				BESTUECKZELLE_1720:
					fb_state_entry.i16_next_step := 40;
			END_CASE
		END_IF

(*=======================================================*)
	35:	(* CAM OUT Y-Achse *)
		IF fb_state_entry.E THEN
			st_drive_cmd_y_achse.enu_cmd := CAM_OUT_SLAVE;
		END_IF

		(*-----------------------Weiterschaltbedingungen----------------------------*)
		IF st_drive_cmd_y_achse.enu_cmd = NO_COMMAND AND NOT fb_state_entry.E THEN
			fb_state_entry.i16_next_step := 40;
		END_IF

(*=======================================================*)
	40:	(* Reglerfreigabe setzen , Reset wird bei Bedarf automatisch ausgeführt*)
		IF fb_state_entry.E THEN
			st_drive_cmd.enu_cmd := POWER_ENABLE;
		END_IF

		(*-----------------------Weiterschaltbedingungen----------------------------*)
		IF st_drive_cmd.enu_cmd = NO_COMMAND THEN
			fb_state_entry.i16_next_step := 50;
		END_IF

(*=======================================================*)
	50:	(* Nullpunktverschiebung ist geschrieben *)
		IF fb_state_entry.E THEN
			st_ctrl_out.b_prebereit := TRUE;
		END_IF

		(*-----------------------Weiterschaltbedingungen----------------------------*)
		IF st_ctrl_in.b_init THEN
			CASE gst_datensatz.st_md.i16_typ_zelle OF
				KEINE_ZELLE:
					;

				BESTUECKZELLE_1700, RASTERFOLIE:
					fb_state_entry.i16_next_step := 60;

				BESTUECKZELLE_1720:
					fb_state_entry.i16_next_step := 95;
			END_CASE
		END_IF

(*=======================================================*)
	60: (* Abfrage der Positionen von Z-Achse und Y-Achse *)

		(*-----------------------Weiterschaltbedingungen----------------------------*)
		IF 	z_achse.NcToPlc.ActPos > ST_MotionFunctionPoints.YZTischMasterPos3 AND
			ABS(y_achse.NcToPlc.ActPos - gst_datensatz.st_md.st_md_y_achse.lr_wt_uebergabepos) > 0.5
			THEN
				(* Y-Achse steht in Kollision mit Antriebskonus des Förderbands *)
				fb_state_entry.i16_next_step := 70;
		ELSE
			i16_kollisionszaehler := 0;
			fb_state_entry.i16_next_step := 80;
		END_IF

(*=======================================================*)
	70: (* Im Wiederhohlungsfall -> Fehler *)
		IF fb_state_entry.E THEN
			i16_kollisionszaehler := i16_kollisionszaehler + 1;
		END_IF

		(*-----------------------Weiterschaltbedingungen----------------------------*)
		IF i16_kollisionszaehler > 1 THEN
			sm_positionsueberwachung := TRUE;
			fb_state_entry.i16_next_step := FEHLER;
		ELSE
			fb_state_entry.i16_next_step := 75;
		END_IF

(*=======================================================*)
	75:	(* Fahre Z-Achse und damit Y-Achse aus der Kollisionsposition *)
		IF fb_state_entry.E THEN
			fb_axis.lr_soll_geschwindigkeit := gst_datensatz.st_wkz.r_auto_z;
			fb_axis.st_position.r_soll := ST_MotionFunctionPoints.YZTischMasterPos3;
			st_drive_cmd.enu_cmd := MOVE_ABSOLUTE;
		END_IF

		(*-----------------------Weiterschaltbedingungen----------------------------*)
		IF st_drive_cmd.enu_cmd = NO_COMMAND THEN
			fb_state_entry.i16_next_step := 80;
		END_IF

(*=======================================================*)
	80: (* Auslesen der Y-Position an der aktuellen Z-Position in der Kurvenscheibe *)
		IF fb_state_entry.E THEN
			fb_axis_y_achse.r_master_position := z_achse.NcToPlc.ActPos;
			st_drive_cmd_y_achse.enu_cmd := READ_SLAVE_DYNAMICS;
		END_IF

		(*-----------------------Weiterschaltbedingungen----------------------------*)
		IF st_drive_cmd_y_achse.enu_cmd = NO_COMMAND AND NOT fb_state_entry.E THEN
			fb_state_entry.i16_next_step := 85;
		END_IF

(*=======================================================*)
	85: (* Starte Y-Achse auf die entsprechende Position in der Kurvenscheibe *)
		IF fb_state_entry.E THEN
			lr_slave_position := fb_axis_y_achse.mc_read_camtable_slave_dynamics.SlavePosition;
			axis_y_achse.st_ctrl.in.b_start := TRUE;
		END_IF

		(*-----------------------Weiterschaltbedingungen----------------------------*)
		IF axis_y_achse.st_ctrl.out.b_fertig AND NOT fb_state_entry.E THEN
			axis_y_achse.st_ctrl.in.b_start := FALSE;
			fb_state_entry.i16_next_step := 90;
		END_IF

(*=======================================================*)
	90:	(* CAM IN Y-Achse *)
		IF fb_state_entry.E THEN
			fb_axis_y_achse.st_camscaling_data.SlaveScaling := 1;
			st_drive_cmd_y_achse.enu_cmd := CAM_IN_SLAVE;
		END_IF

		IF y_achse.NcToPlc.CoupleState = 0 THEN
			st_drive_cmd_y_achse.enu_cmd := CAM_IN_SLAVE;
		END_IF

		(*-----------------------Weiterschaltbedingungen----------------------------*)
		IF st_drive_cmd_y_achse.enu_cmd = NO_COMMAND AND NOT fb_state_entry.E THEN
			fb_state_entry.i16_next_step := 95;
		END_IF

(*=======================================================*)
	95:	(* Fahre Z-Achse auf die WT-Übergabeposition *)
		IF fb_state_entry.E THEN
			fb_axis.lr_soll_geschwindigkeit := gst_datensatz.st_wkz.r_auto_z;
			fb_axis.st_position.r_soll := gst_datensatz.st_md.st_md_z_achse.lr_wt_uebergabepos;
			st_drive_cmd.enu_cmd := MOVE_ABSOLUTE;
		END_IF

		(*-----------------------Weiterschaltbedingungen----------------------------*)
		IF st_drive_cmd.enu_cmd = NO_COMMAND THEN
			fb_state_entry.i16_next_step := BEREIT;
		END_IF

(*=======================================================*)
	BEREIT:
		IF fb_state_entry.E THEN
			st_ctrl_out.b_busy:=FALSE;
			st_ctrl_out.b_bereit := TRUE;
			st_ctrl_out.b_fertig := TRUE;
			bm_rastnasen_1_fehlt := FALSE;
			bm_rastnasen_2_fehlt := FALSE;
			enu_cmd_in:=NO_COMMAND;
		END_IF

		IF NOT gst_datensatz.st_wkz.b_rafo_auto_einf_aktiv THEN
			IF 	gst_datensatz.st_md.i16_typ_zelle = RASTERFOLIE AND
				NOT ST_Rasterfolieneinzug.fb_tof_gls_rafo_ende.Q THEN
				fb_state_entry.i16_next_step := FEHLER;
				sm_keine_rafo_im_einzug:=TRUE;
			END_IF
		END_IF

		(*-----------------------Weiterschaltbedingungen----------------------------*)
		IF fb_r_trig_start.Q  THEN
(*			(* Stoppe WT Wechselzeit *)
			zeit_wt_wechsel := TIME_TO_DWORD(fb_ton_taktzeitmessung_wt_wechsel.ET);
			fb_ton_taktzeitmessung_wt_wechsel.IN := FALSE;
			(* Starte Bestückzeit *)
			fb_ton_taktzeitmessung_bestuecken.IN := TRUE;*)
			fb_Z_Achse_einfahren(b_start:= TRUE, t_zeit=> );
			st_ctrl_out.b_fertig := FALSE;
			st_ctrl_out.b_busy:=TRUE;
			i32_anzahl_rasterfolie:=0;
			fb_state_entry.i16_next_step := 110;
		END_IF

		IF 	fb_r_trig_start_in.Q THEN		(*neu! zum Starten einer Positionierung von einem externen Prg.*)
			st_ctrl_out.b_fertig := FALSE;
			st_ctrl_out.b_busy:=TRUE;
			fb_state_entry.i16_next_step := 102;
		END_IF

(*=======================================================*)
	102:	(*Y Achse abkoppeln*)
		IF 	fb_state_entry.E THEN
			b_start_in:=FALSE;
		END_IF

		IF 	y_achse.NcToPlc.CoupleState > 0 THEN
			st_drive_cmd_y_achse.enu_cmd := CAM_OUT_SLAVE;
		ELSE
			fb_state_entry.i16_next_step := 103;
		END_IF

(*=======================================================*)
	103:
		(*-----------------------Weiterschaltbedingungen----------------------------*)
		IF	enu_cmd_in = NO_COMMAND THEN
			fb_state_entry.i16_next_step := BEREIT;
		ELSIF
			enu_cmd_in = CAM_IN_SLAVE THEN
			fb_state_entry.i16_next_step := 90;		 (* Y Achse Cam In und auf Grundstellung fahren   *)

		ELSE
			fb_state_entry.i16_next_step := 104;
		END_IF

(*=======================================================*)
	104: (* Positioniere Achse  *)
		IF 	fb_state_entry.E THEN
			fb_axis.st_position.r_soll := lr_Achspos_in ;
			fb_axis.lr_soll_geschwindigkeit:=lr_Velo_in;
			st_drive_cmd.enu_cmd := enu_cmd_in;
		END_IF

		(*-----------------------Weiterschaltbedingungen----------------------------*)
		IF 	st_drive_cmd.enu_cmd = NO_COMMAND THEN
			fb_state_entry.i16_next_step := BEREIT;
		END_IF

(*=======================================================*)
	110: (* WT-Tag mit RFID-Lesegerät auslesen *)
		IF fb_state_entry.E THEN
			balluff_tag_reader.st_ctrl.in.b_start_lesen := TRUE;
			balluff_tag_reader.fb.i16_addresse := 0;
			balluff_tag_reader.fb.i16_anzahl_byte := SIZEOF(gst_tag_data);
		END_IF

		(*-----------------------Weiterschaltbedingungen----------------------------*)
		IF balluff_tag_reader.st_ctrl.out.b_fertig AND NOT fb_state_entry.E THEN
			ST_Konvertiere_gelese_TagData();

			IF gst_tag_data.WpcNumber >= 1 AND gst_tag_data.WpcNumber <=50 THEN
				fb_state_entry.i16_next_step := 120;
			ELSE
				(* Fehler: Tagnummer ist nicht im gültigem Bereich *)
				sm_tagnummer_ungueltig := TRUE;
				fb_state_entry.i16_next_step := FEHLER;
			END_IF
		END_IF

		IF fb_state_entry.X THEN
			balluff_tag_reader.st_ctrl.in.b_start_lesen := FALSE;
			fb_ton_wz.IN := FALSE;
		END_IF

(*=======================================================*)
	120: (* Die WPCDaten vom ausgelesenen Tag abfragen *)
		IF fb_state_entry.E THEN
			CASE gst_datensatz.st_md.i16_typ_zelle OF
				KEINE_ZELLE:
					;
	
				BESTUECKZELLE_1700, RASTERFOLIE:
					(* Daten Gültig *)
					IF 	(gst_tag_data.StateParts[0] = PART_NEW OR gst_tag_data.StateParts[0] = PART_OK) OR
						hublift_links.st_config.b_station_aktiv OR visu.b_inbetriebnahme OR NOT gst_datensatz.st_md.b_wt_transport_aktiv
						THEN
							fb_state_entry.i16_next_step := 130;
					ELSE
						(* Einfach durchschleusen: Wir muessen nicht bearbeiten. z.B. für gst_tag_data.State01 = PART_DUMMY *)
						fb_state_entry.i16_next_step := BEREIT;
					END_IF

				BESTUECKZELLE_1720:
					(* Daten Gültig *)
					IF 	(gst_tag_data.StateParts[0] = PART_NEW AND gst_tag_data.StateParts[1] = PART_NEW) OR
						(gst_tag_data.StateParts[0] = PART_OK AND gst_tag_data.StateParts[1] = PART_OK) OR
						hublift_links.st_config.b_station_aktiv OR visu.b_inbetriebnahme OR NOT gst_datensatz.st_md.b_wt_transport_aktiv
						THEN
							fb_state_entry.i16_next_step := 130;
					ELSE
						(* Einfach durchschleusen: Wir muessen nicht bearbeiten *)
						fb_state_entry.i16_next_step := BEREIT;
					END_IF
			END_CASE
		END_IF

(*=======================================================*)
		130:	(* Prüfe Bandfreigabe *)

		(*-----------------------Weiterschaltbedingungen----------------------------*)
		CASE gst_datensatz.st_md.i16_typ_zelle OF
			KEINE_ZELLE:
				;

			BESTUECKZELLE_1700:
				IF 	zyl_bawe_querschub.fb.e_sensor1_eingefahren AND
					((gst_barcode_daten.b_band_links_ok AND gst_barcode_daten.b_band_ID_links_ok) OR
					ST_Virtuelle_Masterachse.b_merker_bandende_links) THEN
					fb_state_entry.i16_next_step := 140;
				ELSIF
					zyl_bawe_querschub.fb.e_sensor1_ausgefahren AND
					((gst_barcode_daten.b_band_rechts_ok AND gst_barcode_daten.b_band_ID_rechts_ok) OR
					ST_Virtuelle_Masterachse.b_merker_bandende_rechts) THEN
					fb_state_entry.i16_next_step := 140;
				ELSE
					sm_keine_bandfreigabe := TRUE;
					fb_state_entry.i16_next_step := 180; 	(*Plle mit NOK beschreiben danach FEHLER*)
				END_IF

			BESTUECKZELLE_1720:
				IF 	(gst_barcode_daten.b_band_ok AND gst_barcode_daten.b_band_ID_links_ok AND gst_barcode_daten.b_band_ID_rechts_ok)  OR
					ST_Virtuelle_Masterachse.b_merker_bandende_rechts OR
					ST_Virtuelle_Masterachse.b_merker_bandende_links THEN
					fb_state_entry.i16_next_step := 140;

				ELSE
					sm_keine_bandfreigabe := TRUE;
					fb_state_entry.i16_next_step := 180; 	(*Plle mit NOK beschreiben danach FEHLER*)
				END_IF

			RASTERFOLIE:
				IF 	gst_barcode_daten.b_band_links_ok THEN
					fb_state_entry.i16_next_step := 140;

				ELSE
					sm_keine_bandfreigabe := TRUE;
					fb_state_entry.i16_next_step := 180; 	(*Plle mit NOK beschreiben danach FEHLER*)
				END_IF

		END_CASE

(*=======================================================*)
	140:	(* Muss das Bestückbild neu von Tag ausgelesen werden? *)


		(*-----------------------Weiterschaltbedingungen----------------------------*)
		IF 	s_alte_artikelnummer = gst_datensatz.st_md.s_aktuelle_artikelnummer AND
			gst_datensatz.st_md.b_wt_transport_aktiv AND
			NOT b_kommt_von_init THEN
			fb_state_entry.i16_next_step := 160;
		ELSE
			fb_state_entry.i16_next_step := 150;
		END_IF

(*=======================================================*)
	150:	(* Bestückbild aus DB von Festplatte einlesen. *)
		IF fb_state_entry.E THEN
			b_kommt_von_init := FALSE;
			gi16_bbgen_auftrag := LESE_BESTUECKBILD; (*und ISK*)
		END_IF

		(*-----------------------Weiterschaltbedingungen----------------------------*)
		IF 	gi16_bbgen_auftrag = KEIN_BB_AUFTRAG THEN
			s_alte_artikelnummer := gst_datensatz.st_md.s_aktuelle_artikelnummer;
			fb_state_entry.i16_next_step := 160;
		END_IF

(*=======================================================*)
	160:	(* Suche nach "Pruef" in Artikelnummer (nur für Rasterfolie) *)

		(*-----------------------Weiterschaltbedingungen----------------------------*)
		CASE gst_datensatz.st_md.i16_typ_zelle OF

			BESTUECKZELLE_1700, BESTUECKZELLE_1720:
				fb_state_entry.i16_next_step := 170;

			RASTERFOLIE:
				IF 	(FIND(gst_datensatz.st_md.s_aktuelle_artikelnummer, 'ruef') > 0 OR			(*es wird nur auf ruef abgefragt, weil das P groß oder klein sein kann*)
					FIND(gst_datensatz.st_md.s_aktuelle_artikelnummer,'erth') > 0)THEN
					fb_state_entry.i16_next_step := 370;	(* nicht Bestücken *)
				ELSE
					fb_state_entry.i16_next_step := 170;
				END_IF

		END_CASE

(*=======================================================*)
	170: (* Prüfe Werkzeugreihenfolge *)
		(* 	3 Fälle:
			1:	- PART_NEW	--->	Wir sind die erste Station
			2:	- PART_OK	--->	Vorgänger hat Station Ok bearbeitet
				-			--->	Prüfe dass diese LastUsedTool in der Liste vor unserer Station steht

			3:	- PART_NOK	-->	Kommt hier gar nicht an, trotzdem Fehler abfangen
				- PART_NO	-->	Kommt hier gar nicht an, trotzdem Fehler abfangen
		*)	
		IF fb_state_entry.E THEN
			CASE gst_datensatz.st_md.i16_typ_zelle OF
				KEINE_ZELLE:
					;

				BESTUECKZELLE_1700, BESTUECKZELLE_1720, RASTERFOLIE:
					IF gst_datensatz.st_md.i16_typ_bestueckmodus<>BESTUECKUNG_MANUAL  AND gst_datensatz.st_md.b_wt_transport_aktiv THEN

						i32_UsedTool:=-1;
						k:=-1;
						FOR k := 0 TO 4 DO      (*Werkzeuggruppen durchsuchen*)
							i:=-1;

							CASE gst_datensatz.st_md.i16_typ_bestueckmodus OF

								BESTUECKUNG_MANUAL:
											;
								BESTUECKUNG_HALBAUTO:

									FOR i := 0 TO MaxNoOfWkz DO
										IF 	gst_bestueckbild_halbauto.s_wkzgruppe[k].s_wkznummer[i] = gst_datensatz.st_md.s_aktuelles_wkz THEN
											i32_UsedTool:=i;
										END_IF
									END_FOR

								BESTUECKUNG_AUTO:

									FOR i := 0 TO MaxNoOfWkz DO
										IF 	gst_bestueckbild.s_wkzgruppe[k].s_wkznummer[i] = gst_datensatz.st_md.s_aktuelles_wkz THEN
											i32_UsedTool:=i;
										END_IF
									END_FOR

								ELSE
									sm_typ_bestueckprogramm_falsch := TRUE;
									fb_state_entry.i16_next_step := FEHLER;
							END_CASE

						END_FOR

						(* ------- Fall 1-------- *)
						IF gst_tag_data.StateParts[0]= PART_NEW THEN
							IF 	i32_UsedTool<>-1 THEN
								gst_tag_data.LastUsedTool := DINT_TO_BYTE(i32_UsedTool);
								fb_state_entry.i16_next_step := 190;
							ELSE
							(* NOk *)
								sm_werkzeugreihenfolge_nicht_io := TRUE;
								fb_state_entry.i16_next_step := 180; 	(*Pille mit NOK beschreiben danach FEHLER*)
							END_IF

						(* ------- Fall 2-------- *)
						ELSIF gst_tag_data.StateParts[0] = PART_OK THEN

							(* Ok *)
							IF 	i32_UsedTool<>-1 AND
							 	gst_tag_data.LastUsedTool < i32_UsedTool AND
								i32_UsedTool < gst_tag_data.LastUsedTool+3 THEN
								gst_tag_data.LastUsedTool := DINT_TO_BYTE(i32_UsedTool);
								fb_state_entry.i16_next_step := 190;
							ELSIF gst_tag_data.LastUsedTool = i32_UsedTool THEN
								fb_state_entry.i16_next_step := BEREIT;	(* nichts tun, ich habe schon bestückt *)
							ELSE
							(* NOk *)
								sm_werkzeugreihenfolge_nicht_io := TRUE;
								fb_state_entry.i16_next_step := 180; 	(*Pille mit NOK beschreiben danach FEHLER*)
							END_IF
						(* ------- Fall 3-------- *)
						ELSE
							sm_werkzeugreihenfolge_nicht_io := TRUE;
							fb_state_entry.i16_next_step := 180; 	(*Pille mit NOK beschreiben danach FEHLER*)
						END_IF
					ELSE
						(* Manuelle BB Anwahl *)
						gst_tag_data.LastUsedTool := 0;
						fb_state_entry.i16_next_step := 190;
					END_IF
			END_CASE
		END_IF

(*=======================================================*)
	180: (* Markiere WT als schlecht, weil Werkzeugreihenfolge nicht passt und Ende mit Fehler. *)
		IF fb_state_entry.E THEN
			ST_Markiere_WT_NIO();
		END_IF

		(*-----------------------Weiterschaltbedingungen----------------------------*)
		IF balluff_tag_reader.st_ctrl.out.b_fertig AND NOT fb_state_entry.E THEN
			(* Ok: Daten wurden auf die Pille geschrieben *)
			balluff_tag_reader.st_ctrl.in.b_start_schreiben := FALSE;
			fb_state_entry.i16_next_step := FEHLER;
		END_IF

(*=======================================================*)
	190:	(* Werkzeugreihenfolge in Ordnung *)

		(*-----------------------Weiterschaltbedingungen----------------------------*)
		CASE gst_datensatz.st_md.i16_typ_zelle OF
			KEINE_ZELLE:
				;

			BESTUECKZELLE_1700, RASTERFOLIE:
				IF 	gst_PersDaten.b_Zelle_nicht_in_Betrieb AND (FIND(gst_datensatz.st_md.s_aktuelle_artikelnummer,'ruef') = 0 AND			(*es wird nur auf ruef abgefragt, weil das P groß oder klein sein kann*)
					FIND(gst_datensatz.st_md.s_aktuelle_artikelnummer,'erth') = 0) THEN
					fb_state_entry.i16_next_step := 195;
				ELSE
					IF 	gst_datensatz.st_md.b_tagreader_fahrend THEN
						fb_state_entry.i16_next_step := 200;
					ELSE
						fb_state_entry.i16_next_step := 210;
					END_IF
				END_IF


				(*Abbruch wenn kein Pin bestückt wird*)
				IF	gst_datensatz.st_bestueckprogramm.i32_anzahl=0 THEN
					fb_state_entry.i16_next_step := 350;
					bm_kein_Pin_im_BB:= TRUE;
					IF FIND(gst_datensatz.st_md.s_aktuelle_artikelnummer,'ruef') = 0 AND			(*es wird nur auf ruef abgefragt, weil das P groß oder klein sein kann*)
						FIND(gst_datensatz.st_md.s_aktuelle_artikelnummer,'erth') = 0THEN
						gst_PersDaten.b_Zelle_nicht_in_Betrieb := TRUE;
					END_IF
				ELSE
					bm_kein_Pin_im_BB:= FALSE;
				END_IF

			BESTUECKZELLE_1720:
				IF 	gst_PersDaten.b_Zelle_nicht_in_Betrieb AND (FIND(gst_datensatz.st_md.s_aktuelle_artikelnummer,'ruef') = 0 AND			(*es wird nur auf ruef abgefragt, weil das P groß oder klein sein kann*)
					FIND(gst_datensatz.st_md.s_aktuelle_artikelnummer,'erth') = 0) THEN
					fb_state_entry.i16_next_step := 395;
				ELSE
					IF gst_datensatz.st_md.	b_tagreader_fahrend THEN
						fb_state_entry.i16_next_step := 400;
					ELSE
						fb_state_entry.i16_next_step := 405;
					END_IF
				END_IF

				(*Abbruch wenn kein Pin bestückt wird*)
				IF	gst_datensatz.st_bestueckprogramm.i32_anzahl=0 THEN
					fb_state_entry.i16_next_step := 460;
					bm_kein_Pin_im_BB:= TRUE;
					IF 	FIND(gst_datensatz.st_md.s_aktuelle_artikelnummer,'ruef') = 0 AND			(*es wird nur auf ruef abgefragt, weil das P groß oder klein sein kann*)
						FIND(gst_datensatz.st_md.s_aktuelle_artikelnummer,'erth') = 0 THEN
						gst_PersDaten.b_Zelle_nicht_in_Betrieb := TRUE;
					END_IF
				ELSE
					bm_kein_Pin_im_BB:= FALSE;
				END_IF
		END_CASE

(*=======================================================*)
	195: (*Warten bis keine ander Produktions Meldung ansteht *)
		IF	TestAndSet(ST_Message_Produktion.LockFlag) THEN
			ST_Message_Produktion.ClearMessageLines();
			fb_state_entry.i16_next_step := 196;
		END_IF

(*=======================================================*)
	196:  (*Produktions Meldung*)
		Visu.MeldungProduktion.Color_R := 255;
		Visu.MeldungProduktion.Color_G := 0;
		Visu.MeldungProduktion.Color_B := 0;
		IF visu.s_akt_sprache = 'de' THEN
			Visu.MeldungProduktion.Name:='Zelle war nicht in Betrieb, bitte Instandhalter informieren!$R$N$R$NÖler,Bestückposition, Seitenversatz und Biegewinkel kontrollieren$R$NMeldung kann nur eingeloggt quittiert werden';
		ELSIF visu.s_akt_sprache = 'en' THEN
			Visu.MeldungProduktion.Name:='Station has not been used for last order, please inform Maintenance Technician!$R$N$R$Ncheck oiler, stich position, left/right and bending angle$R$Nmessage can only be acknowledged when logged in';
		ELSIF visu.s_akt_sprache = 'cz' THEN
			Visu.MeldungProduktion.Name:='Bunka nebyla v provozu, informujte prosim serizovace. Zkontrolujte olej, nastaveni os a uhel ohybu.$R$NZprávu lze potvrdit jen po prihlaseni ';
		END_IF
		Visu.MeldungProduktion.ShowMessage := TRUE;
		Visu.MeldungProduktion.Button1.sichtbar:=TRUE;	(*OK*)
		Visu.MeldungProduktion.Button1.Text:='Ok';

		(*-----------------------Weiterschaltbedingungen----------------------------*)
		IF visu.b_logon THEN
			IF Visu.MeldungProduktion.Button1.tasten THEN
				IF gst_datensatz.st_md.	b_tagreader_fahrend THEN
					fb_state_entry.i16_next_step := 200;
				ELSE
					fb_state_entry.i16_next_step := 210;
				END_IF
			END_IF
		END_IF

		IF fb_state_entry.X THEN
			gst_PersDaten.b_Zelle_nicht_in_Betrieb := FALSE;
		END_IF

(*=======================================================*)
	200:  (* Fahre Z-Achse bis auf 0-Koordinate des ISK - Y-Achse ist gekoppelt *)
		(* Einfahrhöhe der Y-Achse beachten! *)
		IF fb_state_entry.E THEN
			IF gst_datensatz.st_wkz.bFahreSofortAufUebergabePosition THEN
				fb_axis.lr_soll_geschwindigkeit := st_geschwindigkeiten.lr_auto_max;
			ELSE
				fb_axis.lr_soll_geschwindigkeit := gst_datensatz.st_wkz.r_auto_z;
			END_IF
			fb_axis.st_position.r_soll := gst_datensatz.st_isk.lr_pos_z_0 + gst_datensatz.st_wkz.lr_offset_z_pos_0 + gst_datensatz.st_wt.lr_offset_z_pos_0 + gst_datensatz.st_md.lr_offset_z_pos_0 + gst_datensatz.st_bestueckprogramm.lr_z[0];
			st_drive_cmd.enu_cmd := MOVE_ABSOLUTE;
			(*Rasterfolie kann gleich eingezogen werden. Zeitersparnis*)
			IF gst_datensatz.st_md.i16_typ_zelle = RASTERFOLIE THEN
				rasterfolieneinzug.st_ctrl.in.b_start := TRUE;
			END_IF
		END_IF

		(*-----------------------Weiterschaltbedingungen----------------------------*)
		(* Z-Achse losfahren und währenddessen beschreibt der Tagreader die Pille *)
		(*Rasterfolie kann gleich eingezogen werden. Zeitersparnis*)
		IF gst_datensatz.st_md.i16_typ_zelle = RASTERFOLIE THEN
			IF NOT rasterfolieneinzug.st_ctrl.out.b_fertig THEN
				rasterfolieneinzug.st_ctrl.in.b_start := FALSE;
				fb_state_entry.i16_next_step := 210;
			END_IF
		ELSE
			fb_state_entry.i16_next_step := 210;
		END_IF

(*=======================================================*)
	210:	(* WT als schlecht markieren *)
		IF fb_state_entry.E THEN
			ST_Markiere_WT_NIO();
		END_IF

		(*-----------------------Weiterschaltbedingungen----------------------------*)
		IF balluff_tag_reader.st_ctrl.out.b_fertig AND NOT fb_state_entry.E THEN
			(* Ok: Daten sind auf der Pille *)
			balluff_tag_reader.st_ctrl.in.b_start_schreiben := FALSE;
			IF gst_datensatz.st_md.b_tagreader_fahrend THEN
				(* Auf Z-Achse warten *)
				fb_state_entry.i16_next_step := 220;
			ELSE
				(* Daten geschrieben und erst jetzt die Z-Achse fahren *)
				fb_state_entry.i16_next_step := 230;
			END_IF
		END_IF

(*=======================================================*)
	220:	(* Warte noch auf die Z-Achse, bis sie im Ziel steht. *)

		(*-----------------------Weiterschaltbedingungen----------------------------*)
		IF st_drive_cmd.enu_cmd = NO_COMMAND THEN
			IF gst_datensatz.st_md.i16_typ_zelle = RASTERFOLIE THEN
				IF rasterfolieneinzug.st_ctrl.out.b_fertig THEN
					fb_state_entry.i16_next_step := 240;
				END_IF
			ELSE
				fb_state_entry.i16_next_step := 240;
			END_IF
		END_IF

(*=======================================================*)
	230:(* Fahre Z-Achse bis auf 0-Koordinate des ISK - Y-Achse ist gekoppelt *)
		(* Einfahrhöhe der Y-Achse beachten! *)
		IF fb_state_entry.E THEN
			(* Z-Achse verfahren*)
			IF gst_datensatz.st_wkz.bFahreSofortAufUebergabePosition THEN
				fb_axis.lr_soll_geschwindigkeit := st_geschwindigkeiten.lr_auto_max;
			ELSE
				fb_axis.lr_soll_geschwindigkeit := gst_datensatz.st_wkz.r_auto_z;
			END_IF
			fb_axis.st_position.r_soll := gst_datensatz.st_isk.lr_pos_z_0 + gst_datensatz.st_wkz.lr_offset_z_pos_0 + gst_datensatz.st_wt.lr_offset_z_pos_0 + gst_datensatz.st_md.lr_offset_z_pos_0 + gst_datensatz.st_bestueckprogramm.lr_z[0];
			st_drive_cmd.enu_cmd := MOVE_ABSOLUTE;
			(*Rasterfolie kann gleich eingezogen werden. Zeitersparnis*)
			IF gst_datensatz.st_md.i16_typ_zelle = RASTERFOLIE THEN
				rasterfolieneinzug.st_ctrl.in.b_start := TRUE;
			END_IF
		END_IF

		(*-----------------------Weiterschaltbedingungen----------------------------*)
		(* Z-Achse losfahren und währenddessen beschreibt der Tagreader die Pille *)
		(*Rasterfolie kann gleich eingezogen werden. Zeitersparnis*)
		IF gst_datensatz.st_md.i16_typ_zelle = RASTERFOLIE THEN
			IF NOT rasterfolieneinzug.st_ctrl.out.b_fertig THEN
				rasterfolieneinzug.st_ctrl.in.b_start := FALSE;
				fb_state_entry.i16_next_step := 235;
			END_IF
		ELSE
			fb_state_entry.i16_next_step := 235;
		END_IF

(*=======================================================*)
	235:	(* Warte noch auf die Z-Achse, bis sie im Ziel steht. *)

		(*-----------------------Weiterschaltbedingungen----------------------------*)
		IF st_drive_cmd.enu_cmd = NO_COMMAND THEN
			IF gst_datensatz.st_md.i16_typ_zelle = RASTERFOLIE THEN
				IF rasterfolieneinzug.st_ctrl.out.b_fertig THEN
					fb_state_entry.i16_next_step := 240;
				END_IF
			ELSE
				fb_state_entry.i16_next_step := 240;
			END_IF
		END_IF

(*=======================================================*)
	240:	(* Camout Y-Achse *)
		IF fb_state_entry.E THEN
			st_drive_cmd_y_achse.enu_cmd := CAM_OUT_SLAVE;
		END_IF

		(*-----------------------Weiterschaltbedingungen----------------------------*)
		IF st_drive_cmd_y_achse.enu_cmd = NO_COMMAND THEN
			fb_state_entry.i16_next_step := 250;
		END_IF

(*=======================================================*)
	250: (* Start Y-Achse positionieren auf  0-Koordinate  des ISK *)
		IF fb_state_entry.E THEN
			axis_y_achse.st_ctrl.in.b_start := TRUE;
		END_IF

		(*-----------------------Weiterschaltbedingungen----------------------------*)
		IF axis_y_achse.st_ctrl.out.b_fertig THEN	(* axis_y_achse.st_ctrl.out.b_busy  THEN *)
			fb_state_entry.i16_next_step := 255;
		END_IF

		IF fb_state_entry.X THEN
			axis_y_achse.st_ctrl.in.b_start := FALSE;
		END_IF

(*=======================================================*)
	255: (* Start Y-Achse positionieren auf  0-Koordinate  des ISK *)

		(*-----------------------Weiterschaltbedingungen----------------------------*)
		IF 	axis_y_achse.st_ctrl.out.b_fertig  THEN
			fb_state_entry.i16_next_step := 260;
		END_IF

(*=======================================================*)
	260:
		IF fb_state_entry.E THEN
			fb_Z_Achse_einfahren(b_start:= FALSE, t_zeit=> t_Z_Achse_einfahren);
			fb_Bestueckung(b_start:= TRUE, t_zeit=> );
		END_IF

		CASE gst_datensatz.st_md.i16_typ_zelle OF
			KEINE_ZELLE:
				;

			BESTUECKZELLE_1700:
				(* Führung wird an die Bestückachse abgegeben und die Z-Achse und Y-Achse wird ausschliesslich über Kurvenscheiben-Kopplung verfahren *)
				IF fb_state_entry.E THEN
					axis_virt_master.st_ctrl.in.b_start := TRUE;
				END_IF

				(*-----------------------Weiterschaltbedingungen----------------------------*)
				IF NOT axis_virt_master.st_ctrl.out.b_fertig THEN
					axis_virt_master.st_ctrl.in.b_start := FALSE;
					fb_state_entry.i16_next_step := 270;
				END_IF

			RASTERFOLIE:
				(* Starten der Rasterfolienmontagestation *)
				IF fb_state_entry.E THEN
					rasterfolienmontage.st_ctrl.in.b_start := TRUE;
				END_IF

				(*-----------------------Weiterschaltbedingungen----------------------------*)
				IF NOT rasterfolienmontage.st_ctrl.out.b_fertig THEN
					rasterfolienmontage.st_ctrl.in.b_start := FALSE;
					fb_state_entry.i16_next_step := 290;
				END_IF
		END_CASE

(*=======================================================*)
	270:	(* Bestückzelle 1700 *)

		(*-----------------------Weiterschaltbedingungen----------------------------*)
		IF axis_virt_master.st_ctrl.out.b_fertig THEN
			fb_state_entry.i16_next_step := 300;
		END_IF

		IF fb_state_entry.X THEN
			(* Stoppe Bestückzeit *)
			zeit_wt_bestuecken := TIME_TO_DWORD(fb_ton_taktzeitmessung_bestuecken.ET);
			fb_ton_taktzeitmessung_bestuecken.IN := FALSE;

			(* Starte WT Wechselzeit *)
			fb_ton_taktzeitmessung_wt_wechsel.IN := TRUE;
			fb_Bestueckung(b_start:= FALSE, t_zeit=>t_Bestueckung );
			fb_Z_Achse_ausfahren(b_start:= TRUE, t_zeit=> );
		END_IF

(*=======================================================*)
	290:	(* Rasterfolie *)

		(*-----------------------Weiterschaltbedingungen----------------------------*)
		IF 	rasterfolienmontage.st_ctrl.out.b_fertig THEN
			fb_state_entry.i16_next_step := 294;
		END_IF

		IF fb_state_entry.X THEN
			(* Stoppe Bestückzeit *)
			zeit_wt_bestuecken := TIME_TO_DWORD(fb_ton_taktzeitmessung_bestuecken.ET);
			fb_ton_taktzeitmessung_bestuecken.IN := FALSE;
			(* Starte WT Wechselzeit *)
			fb_ton_taktzeitmessung_wt_wechsel.IN := TRUE;
			fb_Bestueckung(b_start:= FALSE, t_zeit=>t_Bestueckung );
			fb_Z_Achse_ausfahren(b_start:= TRUE, t_zeit=> );
		END_IF

(*=======================================================*)
	294:(* Fahre Z-Achse auf  Rasterfolienprüfposition *)
		IF fb_state_entry.E THEN


			(* Z-Achse verfahren*)
			fb_axis.lr_soll_geschwindigkeit := gst_datensatz.st_wkz.r_auto_z;
			fb_axis.st_position.r_soll := 	gst_datensatz.st_isk.lr_pos_z_0 + gst_datensatz.st_wkz.lr_offset_z_pos_0 + gst_datensatz.st_wt.lr_offset_z_pos_0 + gst_datensatz.st_md.lr_offset_z_pos_0 + gst_datensatz.st_bestueckprogramm.lr_z[i32_anzahl_rasterfolie] +	(*Bestückposition*)
										gst_datensatz.st_wkz.st_rasterfolie.lr_pruefpos_rafo;	(*Abstand zwischen Bestückposition und Prüfposition*)
			st_drive_cmd.enu_cmd := MOVE_ABSOLUTE;
		END_IF

		(*-----------------------Weiterschaltbedingungen----------------------------*)
		IF 	st_drive_cmd.enu_cmd = NO_COMMAND AND
			ST_Rasterfolienmontage.arr_rafo_schieberegister[i32_anzahl_rasterfolie] THEN (*Folie vorhanden*)
			fb_state_entry.i16_next_step := 296;
		END_IF

(*=======================================================*)
	296:	(* Anzahl der Rasterfolien prüfen*)

		IF 	fb_state_entry.E THEN
			i32_anzahl_rasterfolie:=i32_anzahl_rasterfolie+1;
		END_IF

		(*-----------------------Weiterschaltbedingungen----------------------------*)
		IF 	i32_anzahl_rasterfolie = gst_datensatz.st_bestueckprogramm.i32_anzahl THEN
			fb_state_entry.i16_next_step := 300;	 (*Ende*)
		ELSE
			fb_state_entry.i16_next_step := 297;	 (*zur nächsten Folie*)
		END_IF

(*=======================================================*)
	297:(* Fahre Z-Achse auf nächste Rasterfolienposition *)
		IF 	fb_state_entry.E THEN
			(* Z-Achse verfahren*)
			fb_axis.lr_soll_geschwindigkeit := gst_datensatz.st_wkz.r_auto_z;
			fb_axis.st_position.r_soll := gst_datensatz.st_isk.lr_pos_z_0 + gst_datensatz.st_wkz.lr_offset_z_pos_0 + gst_datensatz.st_wt.lr_offset_z_pos_0 + gst_datensatz.st_md.lr_offset_z_pos_0 + gst_datensatz.st_bestueckprogramm.lr_z[i32_anzahl_rasterfolie];
			st_drive_cmd.enu_cmd := MOVE_ABSOLUTE;
		END_IF

		(*-----------------------Weiterschaltbedingungen----------------------------*)
		IF st_drive_cmd.enu_cmd = NO_COMMAND THEN
			fb_state_entry.i16_next_step := 298;
		END_IF

(*=======================================================*)
	298:(* Fahre Z-Achse auf nächste Rasterfolienposition *)
		IF 	fb_state_entry.E THEN
			(*Rasterfolie kann gleich eingezogen werden. Zeitersparnis*)
			rasterfolieneinzug.st_ctrl.in.b_start := TRUE;
		END_IF

		(*-----------------------Weiterschaltbedingungen----------------------------*)
		(* Z-Achse losfahren und währenddessen beschreibt der Tagreader die Pille *)
		(*Rasterfolie kann gleich eingezogen werden. Zeitersparnis*)
		IF NOT rasterfolieneinzug.st_ctrl.out.b_fertig THEN
			rasterfolieneinzug.st_ctrl.in.b_start := FALSE;
			fb_state_entry.i16_next_step := 299;
		END_IF

(*=======================================================*)
	299:	(* Neue Folie eingezogen. *)

		(*-----------------------Weiterschaltbedingungen----------------------------*)
		IF rasterfolieneinzug.st_ctrl.out.b_fertig THEN
			fb_state_entry.i16_next_step := 240;	(*zurück zum nächsten Folien setzen*)
		END_IF

(*=======================================================*)
	300: (* Auslesen der Y-Position an der aktuellen Z-Position in der Kurvenscheibe *)
		IF 	fb_state_entry.E THEN
			fb_axis_y_achse.r_master_position := z_achse.NcToPlc.ActPos;
			st_drive_cmd_y_achse.enu_cmd := READ_SLAVE_DYNAMICS;
		END_IF

		(*-----------------------Weiterschaltbedingungen----------------------------*)
		IF 	st_drive_cmd_y_achse.enu_cmd = NO_COMMAND THEN
			fb_state_entry.i16_next_step := 310;
		END_IF

(*=======================================================*)
	310: (* Start Y-Achse positionieren zurück auf die Kurvenbahn *)
		IF 	fb_state_entry.E THEN
			lr_slave_position := fb_axis_y_achse.mc_read_camtable_slave_dynamics.SlavePosition;
			axis_y_achse.st_ctrl.in.b_start_2 := TRUE;
		END_IF

		(*-----------------------Weiterschaltbedingungen----------------------------*)
		IF axis_y_achse.st_ctrl.out.b_fertig_2 AND NOT fb_state_entry.E THEN
			axis_y_achse.st_ctrl.in.b_start_2 := FALSE;
			fb_state_entry.i16_next_step := 315;
		END_IF

(*=======================================================*)
	315: (* Abfrage, ob sofort auf Übergabeposition gefahren werden soll *)

		(*-----------------------Weiterschaltbedingungen----------------------------*)
		IF gst_datensatz.st_wkz.bFahreSofortAufUebergabePosition THEN
			fb_state_entry.i16_next_step := 330;
		ELSE
			fb_state_entry.i16_next_step := 320;
		END_IF

(*=======================================================*)
	320:	(* Fahre Z-Achse bis auf Anfang der Kurvenbahn *)
		IF fb_state_entry.E THEN
			fb_axis.lr_soll_geschwindigkeit := st_geschwindigkeiten.lr_auto_max;
			IF gst_datensatz.st_wkz.b_variable_einfahrposition THEN
				fb_axis.st_position.r_soll := gst_datensatz.st_wkz.st_yz_tisch.r_wkz_einfahrpos_z;
			ELSE
				fb_axis.st_position.r_soll := ST_MotionFunctionPoints.YZTischMasterPos2;
			END_IF
			st_drive_cmd.enu_cmd := MOVE_ABSOLUTE;
		END_IF

		(*-----------------------Weiterschaltbedingungen----------------------------*)
		IF st_drive_cmd.enu_cmd = NO_COMMAND THEN
			fb_state_entry.i16_next_step := 330;
		END_IF

(*=======================================================*)
	330:	(* Camin Y-Achse *)
		IF fb_state_entry.E THEN
			fb_axis_y_achse.st_camscaling_data.SlaveScaling := 1;
			st_drive_cmd_y_achse.enu_cmd := CAM_IN_SLAVE;
		END_IF

		(*-----------------------Weiterschaltbedingungen----------------------------*)
		IF st_drive_cmd_y_achse.enu_cmd = NO_COMMAND THEN
			fb_state_entry.i16_next_step := 340;
		END_IF

(*=======================================================*)
	340:	(* Fahre Z-Achse mit gekoppelter Y-Achse bis auf Übergabeposition *)
		IF fb_state_entry.E THEN
			IF gst_datensatz.st_wkz.bFahreSofortAufUebergabePosition THEN
				fb_axis.lr_soll_geschwindigkeit := st_geschwindigkeiten.lr_auto_max;
			ELSE
				fb_axis.lr_soll_geschwindigkeit := gst_datensatz.st_wkz.r_auto_z;
			END_IF
			fb_axis.st_position.r_soll := gst_datensatz.st_md.st_md_z_achse.lr_wt_uebergabepos;
			st_drive_cmd.enu_cmd := MOVE_ABSOLUTE;
		END_IF

		(*Nach einem Bandwechsel soll nach X-Teilen gestoppt werden.*)
		IF gst_datensatz.st_wkz.i16_anzahl_Teile_autostop_bandwechsel > 0 THEN
			IF gi16_anzahl_Teile_autostop_bandwechsel = gst_datensatz.st_wkz.i16_anzahl_Teile_autostop_bandwechsel THEN
				Teile_nach_Bandwechsel := TRUE;
				gb_nach_bawe_einzelfertigung := TRUE;
			END_IF
		END_IF

		(*-----------------------Weiterschaltbedingungen----------------------------*)
		IF gb_memEndOfBandMarkNIO THEN
			fb_state_entry.i16_next_step := 370;
		ELSE
			IF gst_datensatz.st_md.b_tagreader_fahrend THEN
				(* Pille sofort beschreiben *)
				fb_state_entry.i16_next_step := 350;
			ELSE
				IF st_drive_cmd.enu_cmd = NO_COMMAND THEN
					(* Warte mit Pille beschreiben, bis der Bestücktisch im Ziel ist *)
					fb_state_entry.i16_next_step := 350;
				END_IF
			END_IF
		END_IF


		IF	gst_datensatz.st_md.b_wt_transport_aktiv =FALSE THEN
			visu.b_merker_vollbestuecken:= FALSE;
			s_alte_artikelnummer := '';
			fb_state_entry.i16_next_step := 360;
		END_IF

		IF fb_state_entry.X THEN
			Teile_nach_Bandwechsel:= FALSE;
			IF gst_datensatz.st_wkz.i16_anzahl_Teile_autostop_bandwechsel <> 0 THEN
				gi16_anzahl_Teile_autostop_bandwechsel := gi16_anzahl_Teile_autostop_bandwechsel + 1;
			END_IF
		END_IF

(*=======================================================*)
	350: (* Schreibe Daten auf Tag *)
		IF fb_state_entry.E THEN
			(* Auswertung der Bestückung (Pins bzw. Rasterplatte) des ISK *)
			ST_Markiere_WT_IO();
		END_IF

		(*-----------------------Weiterschaltbedingungen----------------------------*)
		IF balluff_tag_reader.st_ctrl.out.b_fertig AND NOT fb_state_entry.E THEN
			balluff_tag_reader.st_ctrl.in.b_start_schreiben := FALSE;
			fb_state_entry.i16_next_step := 360;
		END_IF

(*=======================================================*)
	360:	(* Aktualisiere letztes benutzes Werkzeug *)
		IF fb_state_entry.E THEN
			ST_Schreibe_LastUsedTool();
		END_IF

		(*-----------------------Weiterschaltbedingungen----------------------------*)
		IF balluff_tag_reader.st_ctrl.out.b_fertig AND NOT fb_state_entry.E THEN
			balluff_tag_reader.st_ctrl.in.b_start_schreiben := FALSE;
			IF gst_datensatz.st_md.b_tagreader_fahrend THEN
				fb_state_entry.i16_next_step := 370;
			ELSE
				fb_state_entry.i16_next_step := 380;
				fb_Z_Achse_ausfahren(b_start:= FALSE, t_zeit=>t_Z_Achse_ausfahren );
			END_IF
		END_IF

(*=======================================================*)
	370:	(* Warte noch auf die Z-Achse, bis sie auf der Übergabeposition steht. *)

		gb_memEndOfBandMarkNIO := FALSE;

		(*-----------------------Weiterschaltbedingungen----------------------------*)
		IF st_drive_cmd.enu_cmd = NO_COMMAND THEN
			fb_state_entry.i16_next_step := 380;
			fb_Z_Achse_ausfahren(b_start:= FALSE, t_zeit=>t_Z_Achse_ausfahren );
		END_IF

(*=======================================================*)
	380:

		CASE gst_datensatz.st_md.i16_typ_zelle OF
			KEINE_ZELLE:
				;

			BESTUECKZELLE_1700:
				(*-----------------------Weiterschaltbedingungen----------------------------*)
				fb_state_entry.i16_next_step := BEREIT;

			RASTERFOLIE:
				(*-----------------------Weiterschaltbedingungen----------------------------*)
				IF rasterfolienmontage.st_ctrl.out.b_fertig_2 THEN
					fb_state_entry.i16_next_step := BEREIT;
				END_IF
		END_CASE

		IF fb_state_entry.X THEN
			(* Stoppe Bestückzeit *)
			zeit_wt_bestuecken := TIME_TO_DWORD(fb_ton_taktzeitmessung_bestuecken.ET);
			fb_ton_taktzeitmessung_bestuecken.IN := FALSE;
			(* Starte WT Wechselzeit *)
			fb_ton_taktzeitmessung_wt_wechsel.IN := TRUE;
		END_IF

(*==========================Bestückzelle1720=============================*)
	395: (*Warten bis keine ander Produktions Meldung ansteht *)
		IF	TestAndSet(ST_Message_Produktion.LockFlag) THEN
			ST_Message_Produktion.ClearMessageLines();
			fb_state_entry.i16_next_step := 396;
		END_IF

(*=======================================================*)
	396:  (*Produktions Meldung*)
		Visu.MeldungProduktion.Color_R := 255;
		Visu.MeldungProduktion.Color_G := 0;
		Visu.MeldungProduktion.Color_B := 0;
		IF visu.s_akt_sprache = 'de' THEN
			Visu.MeldungProduktion.Name:='Zelle war nicht in Betrieb, bitte Instandhalter informieren!$R$N$R$NÖler,Bestückposition, Seitenversatz und Biegewinkel kontrollieren$R$NMeldung kann nur eingeloggt quittiert werden';
		ELSIF visu.s_akt_sprache = 'en' THEN
			Visu.MeldungProduktion.Name:='Station has not been used for last order, please inform Maintenance Technician!$R$N$R$Ncheck oiler, stich position, left/right and bending angle$R$Nmessage can only be acknowledged when logged in';
		ELSIF visu.s_akt_sprache = 'cz' THEN
			Visu.MeldungProduktion.Name:='Bunka nebyla v provozu, informujte prosim serizovace. Zkontrolujte olej, nastaveni os a uhel ohybu.$R$NZprávu lze potvrdit jen po prihlaseni ';
		END_IF
		Visu.MeldungProduktion.ShowMessage := TRUE;
		Visu.MeldungProduktion.Button1.sichtbar:=TRUE;	(*OK*)
		Visu.MeldungProduktion.Button1.Text:='Ok';

		(*-----------------------Weiterschaltbedingungen----------------------------*)
		IF visu.b_logon THEN
			IF Visu.MeldungProduktion.Button1.tasten THEN
				IF gst_datensatz.st_md.	b_tagreader_fahrend THEN
					fb_state_entry.i16_next_step := 400;
				ELSE
					fb_state_entry.i16_next_step := 405;
				END_IF
			END_IF
		END_IF

		IF fb_state_entry.X THEN
			gst_PersDaten.b_Zelle_nicht_in_Betrieb := FALSE;
		END_IF

(*=======================================================*)
	400:	(* Fahre Z-Achse bis auf die erste Bestückposition *)
		IF fb_state_entry.E THEN
			(* Z-Achse verfahren *)
			fb_axis.lr_soll_geschwindigkeit := gst_datensatz.st_wkz.r_auto_z;
			fb_axis.st_position.r_soll := gst_datensatz.st_isk.lr_pos_z_0 + gst_datensatz.st_wkz.lr_offset_z_pos_0 + gst_datensatz.st_wt.lr_offset_z_pos_0 + gst_datensatz.st_md.lr_offset_z_pos_0 + gst_datensatz.st_bestueckprogramm.lr_z[0];
			st_drive_cmd.enu_cmd := MOVE_ABSOLUTE;
		END_IF

		(*-----------------------Weiterschaltbedingungen----------------------------*)
		(* Z-Achse losfahren und währenddessen beschreibt der Tagreader die Pille *)
		fb_state_entry.i16_next_step := 405;

(*=======================================================*)
	405:	(*  WT als schlecht markieren*)
		IF fb_state_entry.E THEN
			ST_Markiere_WT_NIO();
		END_IF

		(*-----------------------Weiterschaltbedingungen----------------------------*)
		IF balluff_tag_reader.st_ctrl.out.b_fertig AND NOT fb_state_entry.E THEN
			(* Ok: Daten sind auf der Pille *)
			balluff_tag_reader.st_ctrl.in.b_start_schreiben := FALSE;
			IF gst_datensatz.st_md.b_tagreader_fahrend THEN
				(* Warte auf Z-Achse *)
				fb_state_entry.i16_next_step := 410;
			ELSE
				(* Daten geschrieben und erst jetzt die Z-Achse fahren *)
				fb_state_entry.i16_next_step := 420;
			END_IF
		END_IF

(*=======================================================*)
	410:	(* Warte noch auf die Z-Achse, bis sie im Ziel steht. *)

		(*-----------------------Weiterschaltbedingungen----------------------------*)
		IF st_drive_cmd.enu_cmd = NO_COMMAND THEN
			fb_state_entry.i16_next_step := 430;
		END_IF

(*=======================================================*)
	420:	(* Fahre Z-Achse bis auf die erste Bestückposition *)
		IF fb_state_entry.E THEN
			(* Z-Achse verfahren *)
			fb_axis.lr_soll_geschwindigkeit := gst_datensatz.st_wkz.r_auto_z;
			fb_axis.st_position.r_soll := gst_datensatz.st_isk.lr_pos_z_0 + gst_datensatz.st_wkz.lr_offset_z_pos_0 + gst_datensatz.st_wt.lr_offset_z_pos_0 + gst_datensatz.st_md.lr_offset_z_pos_0 + gst_datensatz.st_bestueckprogramm.lr_z[0];
			st_drive_cmd.enu_cmd := MOVE_ABSOLUTE;
		END_IF

		(*-----------------------Weiterschaltbedingungen----------------------------*)
		IF st_drive_cmd.enu_cmd = NO_COMMAND THEN
			fb_state_entry.i16_next_step := 430;
		END_IF

(*=======================================================*)
	430:	(* Führung wird an die Bestückachse abgegeben und die Z-Achse wird ausschliesslich über Kurvenscheiben-Kopplung verfahren *)
		IF fb_state_entry.E THEN
			fb_Z_Achse_einfahren(b_start:= FALSE, t_zeit=> t_Z_Achse_einfahren);
			fb_Bestueckung(b_start:= TRUE, t_zeit=> );
			axis_virt_master.st_ctrl.in.b_start := TRUE;

			(* Stoppe WT Wechselzeit *)
			zeit_wt_wechsel := TIME_TO_DWORD(fb_ton_taktzeitmessung_wt_wechsel.ET);
			fb_ton_taktzeitmessung_wt_wechsel.IN := FALSE;

			(* Starte Bestückzeit *)
			fb_ton_taktzeitmessung_bestuecken.IN := TRUE;
		END_IF

		(*-----------------------Weiterschaltbedingungen----------------------------*)
		IF NOT axis_virt_master.st_ctrl.out.b_fertig THEN
			axis_virt_master.st_ctrl.in.b_start := FALSE;
			fb_state_entry.i16_next_step := 440;
		END_IF

		IF fb_state_entry.X THEN
			(* Stoppe Bestückzeit *)
			zeit_wt_bestuecken := TIME_TO_DWORD(fb_ton_taktzeitmessung_bestuecken.ET);
			fb_ton_taktzeitmessung_bestuecken.IN := FALSE;

			(* Starte WT Wechselzeit *)
			fb_ton_taktzeitmessung_wt_wechsel.IN := TRUE;
		END_IF

(*=======================================================*)
	440:	(* Warte auf  Bestückachse fertig mit Pins setzen *)

		(*-----------------------Weiterschaltbedingungen----------------------------*)
		IF axis_virt_master.st_ctrl.out.b_fertig THEN
			fb_state_entry.i16_next_step := 450;
			fb_Bestueckung(b_start:=FALSE, t_zeit=>t_Bestueckung);
			fb_Z_Achse_ausfahren(b_start:= TRUE, t_zeit=> );
		END_IF

(*=======================================================*)
	450: (* Fahre Z-Achse zurück zur Übergabeposition *)
		IF fb_state_entry.E THEN
			 fb_axis.st_position.r_soll := gst_datensatz.st_md.st_md_z_achse.lr_wt_uebergabepos;
			st_drive_cmd.enu_cmd := MOVE_ABSOLUTE;
		END_IF

		(*Nach einem Bandwechsel soll nach X-Teilen gestoppt werden.*)
		IF gst_datensatz.st_wkz.i16_anzahl_Teile_autostop_bandwechsel > 0 THEN
			IF gi16_anzahl_Teile_autostop_bandwechsel = gst_datensatz.st_wkz.i16_anzahl_Teile_autostop_bandwechsel THEN
				gb_nach_bawe_einzelfertigung := TRUE;
			END_IF
		END_IF

		(*-----------------------Weiterschaltbedingungen----------------------------*)
		IF gst_datensatz.st_md.b_tagreader_fahrend THEN
			(* Pille sofort beschreiben *)
			fb_state_entry.i16_next_step := 460;
		ELSE
			IF st_drive_cmd.enu_cmd = NO_COMMAND THEN
				(* Warte mit Pille beschreiben *)
				fb_state_entry.i16_next_step := 460;
			END_IF
		END_IF

		IF	gst_datensatz.st_md.b_wt_transport_aktiv =FALSE THEN
			visu.b_merker_vollbestuecken:= FALSE;
			s_alte_artikelnummer := '';
			fb_state_entry.i16_next_step := 480;
		END_IF

		IF fb_state_entry.X THEN
			IF gst_datensatz.st_wkz.i16_anzahl_Teile_autostop_bandwechsel <> 0 THEN
				gi16_anzahl_Teile_autostop_bandwechsel := gi16_anzahl_Teile_autostop_bandwechsel + 1;
			END_IF
		END_IF

(*=======================================================*)
	460: (* Schreibe Daten auf Tag *)
		IF fb_state_entry.E THEN
			(* WT Hat die Maschine auf regulärem Weg wieder verlassen *)
			ST_Markiere_WT_IO();
		END_IF

		(*-----------------------Weiterschaltbedingungen----------------------------*)
		IF balluff_tag_reader.st_ctrl.out.b_fertig AND NOT fb_state_entry.E THEN
			balluff_tag_reader.st_ctrl.in.b_start_schreiben := FALSE;
			fb_state_entry.i16_next_step := 470;
		END_IF

(*=======================================================*)
	470:	(* aktualisiere letztes benutzes Werkzeug *)
		IF fb_state_entry.E THEN
			ST_Schreibe_LastUsedTool();
		END_IF

		IF balluff_tag_reader.st_ctrl.out.b_fertig AND NOT fb_state_entry.E THEN
			balluff_tag_reader.st_ctrl.in.b_start_schreiben := FALSE;
			IF gst_datensatz.st_md.b_tagreader_fahrend THEN
				fb_state_entry.i16_next_step := 480;
			ELSE
				fb_Z_Achse_ausfahren(b_start:= FALSE, t_zeit=> );
				fb_state_entry.i16_next_step := BEREIT;
			END_IF
		END_IF

(*=======================================================*)
	480:	(* Z-Achse ist fertig positioniert *)

		(*-----------------------Weiterschaltbedingungen----------------------------*)
		IF st_drive_cmd.enu_cmd = NO_COMMAND THEN
			fb_Z_Achse_ausfahren(b_start:= FALSE, t_zeit=> );
			fb_state_entry.i16_next_step := BEREIT;
		END_IF

(*=======================================================*)
	FEHLER:
		IF fb_state_entry.E THEN
			st_ctrl_out.b_fehler := TRUE;
			fb_ton_quitt.IN := FALSE;
			st_ctrl_out.b_busy:=FALSE;
		END_IF

		(*-----------------------Weiterschaltbedingungen----------------------------*)
		IF st_ctrl_in.b_quitt AND NOT fb_state_entry.E THEN
			st_ctrl_out.b_fehler := FALSE;
			st_drive_cmd.enu_cmd := RESET;
			st_drive_cmd_y_achse.enu_cmd := RESET;
			fb_ton_quitt.IN := TRUE;
		END_IF

		IF st_ctrl_in.b_stop AND NOT z_achse.Status.HasBeenStopped THEN
			st_drive_cmd.enu_cmd := STOP_AXIS;
		END_IF

		IF st_ctrl_in.b_halt AND z_achse.Status.Moving THEN
			st_drive_cmd.enu_cmd := HALT_AXIS;
			st_geschwindigkeiten.lr_verzoegerung := lr_decceleration_nothalt;
		END_IF

		IF fb_ton_quitt.Q THEN
			fb_ton_quitt.IN := FALSE;
			fb_state_entry.i16_next_step := INIT;
		END_IF

(*=======================================================*)
	STOP:
		IF fb_state_entry.E THEN
			st_ctrl_out.b_busy:=FALSE;
			IF z_achse.NcToPlc.CoupleState = 0 THEN
				st_drive_cmd.enu_cmd := STOP_AXIS;
			END_IF
		END_IF

		(*-----------------------Weiterschaltbedingungen----------------------------*)
		IF st_drive_cmd.enu_cmd = NO_COMMAND AND z_achse.Status.NotMoving THEN
			fb_state_entry.i16_next_step := STILLSTAND;
		END_IF

(*=======================================================*)
	STILLSTAND:
		IF fb_state_entry.E THEN
			st_drive_cmd.enu_cmd := POWER_DISABLE;
			fb_ton_quitt.IN := FALSE;
		END_IF

		(*-----------------------Weiterschaltbedingungen----------------------------*)
		IF st_ctrl_in.b_quitt AND NOT fb_state_entry.E THEN
			fb_ton_quitt.IN := TRUE;
		END_IF

		IF fb_ton_quitt.Q THEN
			fb_ton_quitt.IN := FALSE;
			fb_state_entry.i16_next_step := INIT;
		END_IF

(*=======================================================*)
	HALT:
		IF fb_state_entry.E THEN
			IF z_achse.NcToPlc.CoupleState = 0 THEN
				st_drive_cmd.enu_cmd := HALT_AXIS;
				st_geschwindigkeiten.lr_verzoegerung := lr_decceleration_nothalt;
			END_IF
			fb_ton_quitt.IN := FALSE;
		END_IF

		(*-----------------------Weiterschaltbedingungen----------------------------*)
		IF st_ctrl_in.b_quitt AND NOT fb_state_entry.E THEN
			fb_ton_quitt.IN := TRUE;
		END_IF

		IF fb_ton_quitt.Q THEN
			fb_ton_quitt.IN := FALSE;
			fb_state_entry.i16_next_step := INIT;
		END_IF

(*=======================================================*)
	HANDRAD:	(* Überprüfe Nullpunktverschiebung des Absolutwertgebers auf Korrektheit *)
		IF fb_state_entry.E THEN
			st_ctrl_out.b_fehler := TRUE;
			fb_axis.i16_nc_parameter_nummer := AxisEncoderOffset;
			st_drive_cmd.enu_cmd := READ_NC_PARAMETER;
		END_IF

		(*-----------------------Weiterschaltbedingungen----------------------------*)
		IF st_drive_cmd.enu_cmd = NO_COMMAND THEN
			IF fb_axis.r_wert_nc_read_parameter = gst_datensatz.st_md.st_md_z_achse.lr_nullpunktverschiebung THEN
				fb_state_entry.i16_next_step := 2040;	(* Jogbetrieb *)
			ELSE
				fb_state_entry.i16_next_step := 2010;	(* Reglerfreigabe nehmen und Nullpunktverschiebung schreiben *)
			END_IF
		END_IF

(*=======================================================*)
	2010:	(* Reglerfreigabe wegnehmen , damit Nullpunktverschiebung geschrieben werden kannt*)
		IF fb_state_entry.E THEN
			st_drive_cmd.enu_cmd := POWER_DISABLE;
		END_IF

		(*-----------------------Weiterschaltbedingungen----------------------------*)
		IF st_drive_cmd.enu_cmd = NO_COMMAND THEN
			fb_state_entry.i16_next_step := 2020;
		END_IF

(*=======================================================*)
	2020:	(* Nullpunktverschiebung hat sich geändert, deshalb erst Null reinschreiben, um keinen Additionsfehler zu machen, *)
			(* weil der Wert der Verschiebung beim Neustart komplett auf die Achse geschrieben wird *)
		IF fb_state_entry.E THEN
			fb_axis.i16_nc_parameter_nummer := AxisEncoderOffset;
			fb_axis.r_wert_nc_write_parameter := 0.0;
			st_drive_cmd.enu_cmd := WRITE_NC_PARAMETER;
		END_IF

		(*-----------------------Weiterschaltbedingungen----------------------------*)
		IF st_drive_cmd.enu_cmd = NO_COMMAND THEN
			fb_state_entry.i16_next_step := 2030;
		END_IF

(*=======================================================*)
	2030:	(* Aktuelle Nullpunktverschiebung des Absolutwertgebers an die Achse senden *)
		IF fb_state_entry.E THEN
			fb_axis.i16_nc_parameter_nummer := AxisEncoderOffset;
			fb_axis.r_wert_nc_write_parameter := gst_datensatz.st_md.st_md_z_achse.lr_nullpunktverschiebung;
			st_drive_cmd.enu_cmd := WRITE_NC_PARAMETER;
		END_IF

		(*-----------------------Weiterschaltbedingungen----------------------------*)
		IF st_drive_cmd.enu_cmd = NO_COMMAND THEN
			fb_state_entry.i16_next_step := 2040;
		END_IF

(*=======================================================*)
	2040:	(* Jogbetrieb *)
		IF fb_state_entry.E THEN
			fb_axis.lr_soll_geschwindigkeit := st_geschwindigkeiten.lr_jog;
		END_IF

		IF ST_Euchner_Handbedienpult.i16_Handrad_delta > 0 THEN
			st_drive_cmd.enu_cmd := JOG_VORWAERTS;
		ELSIF ST_Euchner_Handbedienpult.i16_Handrad_delta < 0 THEN
			st_drive_cmd.enu_cmd := JOG_RUECKWAERTS;
		ELSE
			IF z_achse.Status.Moving THEN
				st_drive_cmd.enu_cmd := JOG_STOP;
			END_IF
		END_IF

		(*-----------------------Weiterschaltbedingungen----------------------------*)
		IF gi16_betriebsart <> HAND OR NOT b_hand_dialog_aktiv THEN
			fb_state_entry.i16_next_step := 2050;
		END_IF

(*=======================================================*)
	2050:
		IF fb_state_entry.E THEN
			st_drive_cmd.enu_cmd := ABORT;
		END_IF

		(*-----------------------Weiterschaltbedingungen----------------------------*)
		IF st_drive_cmd.enu_cmd = NO_COMMAND THEN
			fb_state_entry.i16_next_step := 2060;
		END_IF

(*=======================================================*)
	2060:	(* Reglerfreigabe wegnehmen *)
		IF fb_state_entry.E THEN
			st_drive_cmd.enu_cmd := POWER_DISABLE;
		END_IF

		(*-----------------------Weiterschaltbedingungen----------------------------*)
		IF st_drive_cmd.enu_cmd = NO_COMMAND THEN
			st_ctrl_out.b_fehler := FALSE;
			fb_state_entry.i16_next_step := INIT;
		END_IF

(*=======================================================*)
	NULLPUNKT_SETZEN:
		(* Aktuellen Jog beenden, sonst Probleme beim Softwareendschalter*)
		IF fb_state_entry.E THEN
			st_drive_cmd.enu_cmd := JOG_STOP;
		END_IF

		(*-----------------------Weiterschaltbedingungen----------------------------*)
		IF st_drive_cmd.enu_cmd = NO_COMMAND THEN
			fb_state_entry.i16_next_step := 2505;
		END_IF

(*=======================================================*)
	2505:
		(* 	Lese aktuelle Nullpunkt verschiebung von der Hardware. Der Benutze könnte einen falschen
			Wert eingetragen haben *)
		IF fb_state_entry.E THEN
			fb_axis.i16_nc_parameter_nummer := AxisEncoderOffset;
			st_drive_cmd.enu_cmd := READ_NC_PARAMETER;
		END_IF

		(*-----------------------Weiterschaltbedingungen----------------------------*)
		IF st_drive_cmd.enu_cmd = NO_COMMAND THEN
			gst_datensatz.st_md.st_md_z_achse.lr_nullpunktverschiebung := fb_axis.r_wert_nc_read_parameter;
			fb_state_entry.i16_next_step := 2510;
		END_IF

(*=======================================================*)
	2510:	(* Nullpunktverschiebung berechnen *)
		IF fb_state_entry.E THEN
			lr_pos_ohneverschiebung := axis_z_achse.st_visu.lr_position_ist - gst_datensatz.st_md.st_md_z_achse.lr_nullpunktverschiebung;

			gst_datensatz.st_md.st_md_z_achse.lr_nullpunktverschiebung := - lr_pos_ohneverschiebung;
		END_IF

		(*-----------------------Weiterschaltbedingungen----------------------------*)
		(* Aktiviere den Wert in die Hardware *)
		fb_state_entry.i16_next_step := HANDRAD;

(*=======================================================*)
	INBETRIEBNAHME:	(* Überprüfe Nullpunktverschiebung des Absolutwertgebers auf Korrektheit *)
		IF fb_state_entry.E THEN
			fb_axis.i16_nc_parameter_nummer := AxisEncoderOffset;
			st_drive_cmd.enu_cmd := READ_NC_PARAMETER;
		END_IF

		(*-----------------------Weiterschaltbedingungen----------------------------*)
		IF st_drive_cmd.enu_cmd = NO_COMMAND THEN
			IF fb_axis.r_wert_nc_read_parameter = gst_datensatz.st_md.st_md_z_achse.lr_nullpunktverschiebung THEN
				fb_state_entry.i16_next_step := 5100;	(* Reversiersequenz*)
			ELSE
				fb_state_entry.i16_next_step := 5010;	(* Reglerfreigabe nehmen und Nullpunktverschiebung schreiben *)
			END_IF
		END_IF

(*=======================================================*)
	5010:	(* Reglerfreigabe wegnehmen, damit Nullpunktverschiebung geschrieben werden kannt*)
		IF fb_state_entry.E THEN
			st_drive_cmd.enu_cmd := POWER_DISABLE;
		END_IF

		(*-----------------------Weiterschaltbedingungen----------------------------*)
		IF st_drive_cmd.enu_cmd = NO_COMMAND THEN
			fb_state_entry.i16_next_step := 5020;
		END_IF

(*=======================================================*)
	5020:	(* Nullpunktverschiebung hat sich geändert, deshalb erst Null reinschreiben, um keinen Additionsfehler zu machen, *)
			(* weil der Wert der Verschiebung beim Neustart komplett auf die Achse geschrieben wird *)
		IF fb_state_entry.E THEN
			fb_axis.i16_nc_parameter_nummer := AxisEncoderOffset;
			fb_axis.r_wert_nc_write_parameter := 0.0;
			st_drive_cmd.enu_cmd := WRITE_NC_PARAMETER;
		END_IF

		(*-----------------------Weiterschaltbedingungen----------------------------*)
		IF st_drive_cmd.enu_cmd = NO_COMMAND THEN
			fb_state_entry.i16_next_step := 5030;
		END_IF

(*=======================================================*)
	5030:	(* Aktuelle Nullpunktverschiebung des Absolutwertgebers an die Achse senden *)
		IF fb_state_entry.E THEN
			fb_axis.i16_nc_parameter_nummer := AxisEncoderOffset;
			fb_axis.r_wert_nc_write_parameter := gst_datensatz.st_md.st_md_z_achse.lr_nullpunktverschiebung;
			st_drive_cmd.enu_cmd := WRITE_NC_PARAMETER;
		END_IF

		(*-----------------------Weiterschaltbedingungen----------------------------*)
		IF st_drive_cmd.enu_cmd = NO_COMMAND THEN
			fb_state_entry.i16_next_step := 5100;
		END_IF

(*=======================================================*)
	5100:	(* Verfahren der Achse zwischen zwei Punkten zum Testen verschiedener Achsparameter *)
		IF fb_state_entry.E THEN
			fb_axis.lr_soll_geschwindigkeit := st_geschwindigkeiten.lr_jog;
			fb_axis.st_position.lr_ibn_pos_start := 10.0;
			fb_axis.st_position.lr_ibn_pos_ziel := -10.0;
		END_IF

		(*-----------------------Weiterschaltbedingungen----------------------------*)
		IF st_ctrl_in.b_ibn_start THEN
			fb_state_entry.i16_next_step := 5110;
		END_IF

(*=======================================================*)
	5110: (* Fahre Z-Achse auf Startposition *)
(*
		IF fb_state_entry.E THEN
			 fb_axis.st_position.r_soll := fb_axis.st_position.lr_ibn_pos_start;
			st_drive_cmd.enu_cmd := MOVE_ABSOLUTE;
		END_IF

		(*-----------------------Weiterschaltbedingungen----------------------------*)
		IF st_drive_cmd.enu_cmd = NO_COMMAND THEN
			fb_state_entry.i16_next_step := 5120;
		END_IF
*)
		IF fb_state_entry.E THEN
			st_drive_cmd.enu_cmd := POWER_ENABLE;
		END_IF

		(*-----------------------Weiterschaltbedingungen----------------------------*)
		IF st_drive_cmd.enu_cmd = NO_COMMAND THEN
			;
		END_IF

(*=======================================================*)
	5120: (* Pause *)
		IF fb_state_entry.E THEN
			fb_ton_wz.PT := t#500ms;
			fb_ton_wz.IN := TRUE;
		END_IF

		(*-----------------------Weiterschaltbedingungen----------------------------*)
		IF fb_ton_wz.Q THEN
			fb_ton_wz.IN := FALSE;
			fb_state_entry.i16_next_step := 5130;
		END_IF

(*=======================================================*)
	5130: (* Fahre Z-Achse auf Zielposition *)
		IF fb_state_entry.E THEN
			 fb_axis.st_position.r_soll := fb_axis.st_position.lr_ibn_pos_ziel;
			st_drive_cmd.enu_cmd := MOVE_ABSOLUTE;
		END_IF

		(*-----------------------Weiterschaltbedingungen----------------------------*)
		IF st_drive_cmd.enu_cmd = NO_COMMAND THEN
			fb_state_entry.i16_next_step := 5140;
		END_IF

(*=======================================================*)
	5140: (* Pause *)
		IF fb_state_entry.E THEN
			fb_ton_wz.PT := t#500ms;
			fb_ton_wz.IN := TRUE;
		END_IF

		(*-----------------------Weiterschaltbedingungen----------------------------*)
		IF fb_ton_wz.Q THEN
			fb_ton_wz.IN := FALSE;
			fb_state_entry.i16_next_step := 5100;
		END_IF
END_CASE

fb_state_entry(
	i16_next_step:= ,
	i16_pos:= 2,
	s_debugtext:= ,
	E=> ,
	X=> ,
	i16_step=> ,
	i16_last_step=> );

IF st_config_achse.b_config_fertig THEN
	(* Fehlermeldungen und Betriebsmeldungen ab dem Startindex in die globalen Meldungsarrays schreiben *)
	garr_stoermeldungen[st_config_achse.i16_meld_startindex + 0] := st_sm.b_achse_nicht_bb;
	garr_stoermeldungen[st_config_achse.i16_meld_startindex + 1] := st_sm.b_achse_nicht_referenziert;
	garr_stoermeldungen[st_config_achse.i16_meld_startindex + 2] := st_sm.b_keine_verfahrfreigabe;
	garr_stoermeldungen[st_config_achse.i16_meld_startindex + 3] := st_sm.b_achse_nicht_auf_startpos;
	garr_stoermeldungen[st_config_achse.i16_meld_startindex + 4] := st_sm.b_ende_skalierungs_nocke;
	garr_stoermeldungen[st_config_achse.i16_meld_startindex + 5] := st_sm.b_ende_camming_nocke;
	garr_stoermeldungen[st_config_achse.i16_meld_startindex + 6] := st_sm.b_skalierung_noch_aktiv;
	garr_stoermeldungen[st_config_achse.i16_meld_startindex + 7] := FALSE;
	garr_stoermeldungen[st_config_achse.i16_meld_startindex + 8] := FALSE;
	garr_stoermeldungen[st_config_achse.i16_meld_startindex + 9] := FALSE;
	garr_stoermeldungen[st_config_achse.i16_meld_startindex + 10] := sm_positionsueberwachung;
	garr_stoermeldungen[st_config_achse.i16_meld_startindex + 11] := sm_werkzeugreihenfolge_nicht_io;
	garr_stoermeldungen[st_config_achse.i16_meld_startindex + 12] := sm_keine_bandfreigabe;
	garr_stoermeldungen[st_config_achse.i16_meld_startindex + 13] := sm_tagnummer_ungueltig;
	garr_stoermeldungen[st_config_achse.i16_meld_startindex + 14] := FALSE;
	garr_stoermeldungen[st_config_achse.i16_meld_startindex + 15] := sm_typ_bestueckprogramm_falsch;
	garr_stoermeldungen[st_config_achse.i16_meld_startindex + 16] := st_drive_cmd.meldungen.sm_write_soe_parameter;
	garr_stoermeldungen[st_config_achse.i16_meld_startindex + 17] := st_drive_cmd.meldungen.sm_read_soe_parameter;
	garr_stoermeldungen[st_config_achse.i16_meld_startindex + 18] := st_drive_cmd.meldungen.sm_write_nc_parameter;
	garr_stoermeldungen[st_config_achse.i16_meld_startindex + 19] := st_drive_cmd.meldungen.sm_read_nc_parameter;
	garr_stoermeldungen[st_config_achse.i16_meld_startindex + 20] := st_drive_cmd.meldungen.sm_power_enable;
	garr_stoermeldungen[st_config_achse.i16_meld_startindex + 21] := st_drive_cmd.meldungen.sm_power_disable;
	garr_stoermeldungen[st_config_achse.i16_meld_startindex + 22] := st_drive_cmd.meldungen.sm_reset;
	garr_stoermeldungen[st_config_achse.i16_meld_startindex + 23] := st_drive_cmd.meldungen.sm_home;
	garr_stoermeldungen[st_config_achse.i16_meld_startindex + 24] := st_drive_cmd.meldungen.sm_setposition;
	garr_stoermeldungen[st_config_achse.i16_meld_startindex + 25] := st_drive_cmd.meldungen.sm_jog_vorwaerts;
	garr_stoermeldungen[st_config_achse.i16_meld_startindex + 26] := st_drive_cmd.meldungen.sm_jog_rueckwaerts;
	garr_stoermeldungen[st_config_achse.i16_meld_startindex + 27] := st_drive_cmd.meldungen.sm_move_absolute;
	garr_stoermeldungen[st_config_achse.i16_meld_startindex + 28] := st_drive_cmd.meldungen.sm_move_relative;
	garr_stoermeldungen[st_config_achse.i16_meld_startindex + 29] := st_drive_cmd.meldungen.sm_move_velocity;
	garr_stoermeldungen[st_config_achse.i16_meld_startindex + 30] := st_drive_cmd.meldungen.sm_move_modulo;
	garr_stoermeldungen[st_config_achse.i16_meld_startindex + 31] := st_drive_cmd.meldungen.sm_stop_axis;
	garr_stoermeldungen[st_config_achse.i16_meld_startindex + 32] := st_drive_cmd.meldungen.sm_halt_axis;
	garr_stoermeldungen[st_config_achse.i16_meld_startindex + 33] := st_drive_cmd.meldungen.sm_motion_command_timeout;
	garr_stoermeldungen[st_config_achse.i16_meld_startindex + 34] := st_sm.b_achsfehler;
	garr_stoermeldungen[st_config_achse.i16_meld_startindex + 35] := st_sm.b_devicefehler;
	garr_stoermeldungen[st_config_achse.i16_meld_startindex + 36] := st_drive_cmd.meldungen.sm_limit_positiv_erreicht;
	garr_stoermeldungen[st_config_achse.i16_meld_startindex + 37] := st_drive_cmd.meldungen.sm_limit_negativ_erreicht;
	garr_stoermeldungen[st_config_achse.i16_meld_startindex + 38] := st_drive_cmd.meldungen.sm_ec_coe_sdo_write_ex;
	garr_stoermeldungen[st_config_achse.i16_meld_startindex + 39] := st_drive_cmd.meldungen.sm_ec_coe_sdo_read_ex;
	garr_stoermeldungen[st_config_achse.i16_meld_startindex + 40] := st_drive_cmd_y_achse.meldungen.sm_gear_in_slave;
	garr_stoermeldungen[st_config_achse.i16_meld_startindex + 41] := st_drive_cmd_y_achse.meldungen.sm_gear_out_slave;
	garr_stoermeldungen[st_config_achse.i16_meld_startindex + 42] := st_drive_cmd_y_achse.meldungen.sm_cam_in_slave;
	garr_stoermeldungen[st_config_achse.i16_meld_startindex + 43] := st_drive_cmd_y_achse.meldungen.sm_cam_out_slave;
	garr_stoermeldungen[st_config_achse.i16_meld_startindex + 44] := st_drive_cmd_y_achse.meldungen.sm_cam_scaleing_slave;
	garr_stoermeldungen[st_config_achse.i16_meld_startindex + 45] := st_drive_cmd_y_achse.meldungen.sm_camgear_command_timeout;;
	garr_stoermeldungen[st_config_achse.i16_meld_startindex + 46] := st_drive_cmd_y_achse.meldungen.sm_read_motion_funktion_point;
	garr_stoermeldungen[st_config_achse.i16_meld_startindex + 47] := st_drive_cmd_y_achse.meldungen.sm_write_motion_funktion_point;
	garr_stoermeldungen[st_config_achse.i16_meld_startindex + 48] := st_drive_cmd_y_achse.meldungen.sm_read_camtable_slave_dynamics;
	garr_stoermeldungen[st_config_achse.i16_meld_startindex + 49] := st_drive_cmd_y_achse.meldungen.sm_read_camtable_charakteristik;
	garr_stoermeldungen[st_config_achse.i16_meld_startindex + 50] := FALSE;
	garr_stoermeldungen[st_config_achse.i16_meld_startindex + 51] := FALSE;
	garr_stoermeldungen[st_config_achse.i16_meld_startindex + 52] := FALSE;
	garr_stoermeldungen[st_config_achse.i16_meld_startindex + 53] := FALSE;
	garr_stoermeldungen[st_config_achse.i16_meld_startindex + 54] := FALSE;
	garr_stoermeldungen[st_config_achse.i16_meld_startindex + 55] := FALSE;
	garr_stoermeldungen[st_config_achse.i16_meld_startindex + 56] := FALSE;
	garr_stoermeldungen[st_config_achse.i16_meld_startindex + 57] := FALSE;
	garr_stoermeldungen[st_config_achse.i16_meld_startindex + 58] := FALSE;
	garr_stoermeldungen[st_config_achse.i16_meld_startindex + 59] := FALSE;
	garr_stoermeldungen[st_config_achse.i16_meld_startindex + 60] := FALSE;
	garr_stoermeldungen[st_config_achse.i16_meld_startindex + 61] := FALSE;
	garr_stoermeldungen[st_config_achse.i16_meld_startindex + 62] := FALSE;
	garr_stoermeldungen[st_config_achse.i16_meld_startindex + 63] := FALSE;
	garr_stoermeldungen[st_config_achse.i16_meld_startindex + 64] := FALSE;
	garr_stoermeldungen[st_config_achse.i16_meld_startindex + 65] := FALSE;
	garr_stoermeldungen[st_config_achse.i16_meld_startindex + 66] := FALSE;
	garr_stoermeldungen[st_config_achse.i16_meld_startindex + 67] := FALSE;
	garr_stoermeldungen[st_config_achse.i16_meld_startindex + 68] := FALSE;
	garr_stoermeldungen[st_config_achse.i16_meld_startindex + 69] := FALSE;
	garr_stoermeldungen[st_config_achse.i16_meld_startindex + 70] := FALSE;
	garr_stoermeldungen[st_config_achse.i16_meld_startindex + 71] := FALSE;
	garr_stoermeldungen[st_config_achse.i16_meld_startindex + 72] := FALSE;
	garr_stoermeldungen[st_config_achse.i16_meld_startindex + 73] := FALSE;
	garr_stoermeldungen[st_config_achse.i16_meld_startindex + 74] := FALSE;
	garr_stoermeldungen[st_config_achse.i16_meld_startindex + 75] := FALSE;
	garr_stoermeldungen[st_config_achse.i16_meld_startindex + 76] := FALSE;
	garr_stoermeldungen[st_config_achse.i16_meld_startindex + 77] := FALSE;
	garr_stoermeldungen[st_config_achse.i16_meld_startindex + 78] := FALSE;
	garr_stoermeldungen[st_config_achse.i16_meld_startindex + 79] := FALSE;
	garr_stoermeldungen[st_config_achse.i16_meld_startindex + 80] := FALSE;
	garr_stoermeldungen[st_config_achse.i16_meld_startindex + 81] := FALSE;
	garr_stoermeldungen[st_config_achse.i16_meld_startindex + 82] := FALSE;
	garr_stoermeldungen[st_config_achse.i16_meld_startindex + 83] := FALSE;
	garr_stoermeldungen[st_config_achse.i16_meld_startindex + 84] := FALSE;
	garr_stoermeldungen[st_config_achse.i16_meld_startindex + 85] := FALSE;
	garr_stoermeldungen[st_config_achse.i16_meld_startindex + 86] := FALSE;
	garr_stoermeldungen[st_config_achse.i16_meld_startindex + 87] := FALSE;
	garr_stoermeldungen[st_config_achse.i16_meld_startindex + 88] := FALSE;
	garr_stoermeldungen[st_config_achse.i16_meld_startindex + 89] := FALSE;
	garr_stoermeldungen[st_config_achse.i16_meld_startindex + 90] := FALSE;
	garr_stoermeldungen[st_config_achse.i16_meld_startindex + 91] := FALSE;
	garr_stoermeldungen[st_config_achse.i16_meld_startindex + 92] := FALSE;
	garr_stoermeldungen[st_config_achse.i16_meld_startindex + 93] := FALSE;
	garr_stoermeldungen[st_config_achse.i16_meld_startindex + 94] := FALSE;
	garr_stoermeldungen[st_config_achse.i16_meld_startindex + 95] := FALSE;
	garr_stoermeldungen[st_config_achse.i16_meld_startindex + 96] := FALSE;
	garr_stoermeldungen[st_config_achse.i16_meld_startindex + 97] := FALSE;
	garr_stoermeldungen[st_config_achse.i16_meld_startindex + 98] := FALSE;
	garr_stoermeldungen[st_config_achse.i16_meld_startindex + 99] := FALSE;
	
	garr_betriebsmeldungen[st_config_achse.i16_meld_startindex + 0] := bm_kein_Pin_im_BB;
	garr_betriebsmeldungen[st_config_achse.i16_meld_startindex + 1] := bm_rastnasen_1_fehlt;
	garr_betriebsmeldungen[st_config_achse.i16_meld_startindex + 2] := bm_rastnasen_2_fehlt;
	garr_betriebsmeldungen[st_config_achse.i16_meld_startindex + 3] := FALSE;
	garr_betriebsmeldungen[st_config_achse.i16_meld_startindex + 4] := FALSE;
	garr_betriebsmeldungen[st_config_achse.i16_meld_startindex + 5] := FALSE;
	garr_betriebsmeldungen[st_config_achse.i16_meld_startindex + 6] := FALSE;
	garr_betriebsmeldungen[st_config_achse.i16_meld_startindex + 7] := FALSE;
	garr_betriebsmeldungen[st_config_achse.i16_meld_startindex + 8] := FALSE;
	garr_betriebsmeldungen[st_config_achse.i16_meld_startindex + 9] := FALSE;
	garr_betriebsmeldungen[st_config_achse.i16_meld_startindex + 10] := FALSE;
	garr_betriebsmeldungen[st_config_achse.i16_meld_startindex + 11] := FALSE;
	garr_betriebsmeldungen[st_config_achse.i16_meld_startindex + 12] := FALSE;
	garr_betriebsmeldungen[st_config_achse.i16_meld_startindex + 13] := FALSE;
	garr_betriebsmeldungen[st_config_achse.i16_meld_startindex + 14] := FALSE;
	garr_betriebsmeldungen[st_config_achse.i16_meld_startindex + 15] := FALSE;
	garr_betriebsmeldungen[st_config_achse.i16_meld_startindex + 16] := FALSE;
	garr_betriebsmeldungen[st_config_achse.i16_meld_startindex + 17] := FALSE;
	garr_betriebsmeldungen[st_config_achse.i16_meld_startindex + 18] := FALSE;
	garr_betriebsmeldungen[st_config_achse.i16_meld_startindex + 19] := FALSE;
	garr_betriebsmeldungen[st_config_achse.i16_meld_startindex + 20] := FALSE;
	garr_betriebsmeldungen[st_config_achse.i16_meld_startindex + 21] := FALSE;
	garr_betriebsmeldungen[st_config_achse.i16_meld_startindex + 22] := FALSE;
	garr_betriebsmeldungen[st_config_achse.i16_meld_startindex + 23] := FALSE;
	garr_betriebsmeldungen[st_config_achse.i16_meld_startindex + 24] := FALSE;
	garr_betriebsmeldungen[st_config_achse.i16_meld_startindex + 25] := FALSE;
	garr_betriebsmeldungen[st_config_achse.i16_meld_startindex + 26] := FALSE;
	garr_betriebsmeldungen[st_config_achse.i16_meld_startindex + 27] := FALSE;
	garr_betriebsmeldungen[st_config_achse.i16_meld_startindex + 28] := FALSE;
	garr_betriebsmeldungen[st_config_achse.i16_meld_startindex + 29] := FALSE;
	garr_betriebsmeldungen[st_config_achse.i16_meld_startindex + 30] := FALSE;
	garr_betriebsmeldungen[st_config_achse.i16_meld_startindex + 31] := FALSE;
	garr_betriebsmeldungen[st_config_achse.i16_meld_startindex + 32] := FALSE;
	garr_betriebsmeldungen[st_config_achse.i16_meld_startindex + 33] := FALSE;
	garr_betriebsmeldungen[st_config_achse.i16_meld_startindex + 34] := FALSE;
	garr_betriebsmeldungen[st_config_achse.i16_meld_startindex + 35] := FALSE;
	garr_betriebsmeldungen[st_config_achse.i16_meld_startindex + 36] := FALSE;
	garr_betriebsmeldungen[st_config_achse.i16_meld_startindex + 37] := FALSE;
	garr_betriebsmeldungen[st_config_achse.i16_meld_startindex + 38] := FALSE;
	garr_betriebsmeldungen[st_config_achse.i16_meld_startindex + 39] := FALSE;
	garr_betriebsmeldungen[st_config_achse.i16_meld_startindex + 40] := FALSE;
	garr_betriebsmeldungen[st_config_achse.i16_meld_startindex + 41] := FALSE;
	garr_betriebsmeldungen[st_config_achse.i16_meld_startindex + 42] := FALSE;
	garr_betriebsmeldungen[st_config_achse.i16_meld_startindex + 43] := FALSE;
	garr_betriebsmeldungen[st_config_achse.i16_meld_startindex + 44] := FALSE;
	garr_betriebsmeldungen[st_config_achse.i16_meld_startindex + 45] := FALSE;
	garr_betriebsmeldungen[st_config_achse.i16_meld_startindex + 46] := FALSE;
	garr_betriebsmeldungen[st_config_achse.i16_meld_startindex + 47] := FALSE;
	garr_betriebsmeldungen[st_config_achse.i16_meld_startindex + 48] := FALSE;
	garr_betriebsmeldungen[st_config_achse.i16_meld_startindex + 49] := FALSE;
END_IF
END_PROGRAM

(* POU EPT Lib/Achsen/BECKHOFF/ST_AxisJobCtrl_Cam_Gear, ST *)
FUNCTION_BLOCK ST_AxisJobCtrl_Cam_Gear
VAR_INPUT
	r_getriebefaktor						: LREAL;
	r_master_position					: LREAL;
	mc_activation_mode_camin			: MC_CamActivationMode;
	lr_activation_position_camin			: LREAL := 0.0;
	mc_activation_mode_scaleing		: MC_CamActivationMode;
	lr_activation_position_scaleing		: LREAL := 0.0;
	mc_buffermode_axis					: MC_BufferMode;     (*	MC_Aborting,	->sofortiger Abbruch der momentanen Bewegung, bei einem neuen Verfahrbefehl
														MC_Buffered,
														MC_BlendingLow,
														MC_BlendingPrevious,
														MC_BlendingNext,
														MC_BlendingHigh *)
	mc_cam_point_id						: MC_MotionFunctionPoint_ID; (* MC_MotionFunctionPoint_ID : UDINT; *)
	mc_motion_function_point				: MC_MotionFunctionPoint;	(*TYPE MC_MotionFunctionPoint :
																	STRUCT
																	    PointIndex        : MC_MotionFunctionPoint_ID;
																	    FunctionType      : MC_MotionFunctionType;
																	    PointType         : MC_MotionPointType;
																	    RelIndexNextPoint : MC_MotionFunctionPoint_ID;
																	    MasterPos         : LREAL; (* X *)
																	    SlavePos          : LREAL; (* Y *)
																	    SlaveVelo         : LREAL; (* Y' *)
																	    SlaveAcc          : LREAL; (* Y'' *)
																	    SlaveJerk         : LREAL; (* Y''' *)
																	END_STRUCT
																END_TYPE*)
	st_camin_options						: ST_CamInOptions_V2;
	st_camexchange_options				: ST_CamExchangeOptions ;
	mc_cam_table_id					 	: MC_CAM_ID;	(* MC_CAM_ID : UDINT; *)
	mc_reference_cam_table_id				: MC_CAM_ID;	(* MC_CAM_ID : UDINT; *)
	st_camscaling_data						: ST_CamScalingData;	(*STRUCT
																	(* scaling of the X axis of the cam (master scaling) *)
																	MasterScalingMode 	: MC_CamScalingMode;
																	MasterRelative 	: BOOL;
																	MasterOffset 	: LREAL; (* E *)
																	MasterScaling 	: LREAL := 1.0; (* E *)
																
																	(* scaling of the Y axis of the cam (slave scaling) *)
																	SlaveScalingMode 	: MC_CamScalingMode;
																	SlaveRelative 	: BOOL;
																	SlaveOffset 	: LREAL; (* E *)
																	SlaveScaling 	: LREAL := 1.0; (* E *)
																	END_STRUCT*)
END_VAR
VAR_IN_OUT
	st_masterachse						: AXIS_REF;
	st_slaveachse 						: AXIS_REF;
	st_ecd_cmd							: struct_ecd_cmd;
END_VAR
VAR
	fb_ton_cmd_timeout					: TON;
	fb_ton_vz							: TON;
	mc_gearindyn_axis 					: MC_GearInDyn;
	mc_gearout_axis						: MC_GearOut;
	mc_camin_axis						: MC_CamIn_V2;
	mc_camout_axis						: MC_CamOut;
	mc_cam_scaleing						: MC_CamScaling_V2;
	mc_read_motion_function_point			: MC_ReadMotionFunctionPoint;
	mc_write_motion_function_point			: MC_WriteMotionFunctionPoint;
	mc_read_camtable_slave_dynamics		: MC_ReadCamTableSlaveDynamics;
	st_cam_table_characteristics			: MC_TableCharacValues;
	mc_read_camtable_characteristics		: MC_ReadCamTableCharacteristics;
	err_id								: DWORD := 0;
	fb_state_entry							: ST_StateEntry;
	fb_cmd_history						: ST_CommandHistory;
END_VAR
(* Zeiten *)
fb_ton_cmd_timeout(IN:= , PT:= t#5s, Q=> , ET=> );
fb_ton_vz(IN:= , PT:= , Q=> , ET=> );

(* ======================================Schrittkette Drivebefehle======================================== *)
fb_state_entry(
	i16_next_step:= ,
	i16_pos:= 1,
	s_debugtext:= ,
	E=> ,
	X=> ,
	i16_step=> ,
	i16_last_step=> );

CASE fb_state_entry.i16_step OF
(*=======================================================*)
	0:	(* *)
		st_ecd_cmd.enu_cmd := NO_COMMAND;
		st_ecd_cmd.b_job_fehler := FALSE;
		mc_gearindyn_axis.Enable := FALSE;
		mc_gearout_axis.Execute := FALSE;
		mc_camin_axis.Execute := FALSE;
		mc_camout_axis.Execute := FALSE;
		mc_cam_scaleing.Execute := FALSE;
		mc_read_motion_function_point.Execute := FALSE;
		mc_write_motion_function_point.Execute := FALSE;
		mc_read_camtable_slave_dynamics.Execute := FALSE;
		mc_read_camtable_characteristics.Execute := FALSE;
		st_ecd_cmd.meldungen.sm_gear_in_slave := FALSE;
		st_ecd_cmd.meldungen.sm_gear_out_slave := FALSE;
		st_ecd_cmd.meldungen.sm_cam_in_slave := FALSE;
		st_ecd_cmd.meldungen.sm_cam_out_slave := FALSE;
		st_ecd_cmd.meldungen.sm_cam_scaleing_slave := FALSE;
		st_ecd_cmd.meldungen.sm_write_motion_funktion_point := FALSE;
		st_ecd_cmd.meldungen.sm_read_motion_funktion_point := FALSE;
		st_ecd_cmd.meldungen.sm_read_camtable_slave_dynamics := FALSE;
		st_ecd_cmd.meldungen.sm_read_camtable_charakteristik := FALSE;
		st_ecd_cmd.meldungen.sm_camgear_command_timeout := FALSE;

		fb_ton_cmd_timeout.IN := FALSE;
		fb_state_entry.i16_next_step := 10;

(*=======================================================*)
	10:	(* Warte auf Kommando *)
		IF fb_state_entry.E THEN
			st_ecd_cmd.b_job_fehler := FALSE;
			st_ecd_cmd.enu_cmd := NO_COMMAND;
		END_IF

		IF st_ecd_cmd.enu_cmd > NO_COMMAND THEN
			(* Diese Kommandos werden mit Direktsprung ausgeführt, um Zykluszeit zu sparen *)
			IF st_ecd_cmd.enu_cmd = GEAR_IN_SLAVE THEN
				fb_state_entry.i16_next_step := 20;
			ELSIF st_ecd_cmd.enu_cmd = GEAR_OUT_SLAVE THEN
				fb_state_entry.i16_next_step := 30;
			ELSIF st_ecd_cmd.enu_cmd = CAM_IN_SLAVE THEN
				fb_state_entry.i16_next_step := 40;
			ELSIF st_ecd_cmd.enu_cmd = CAM_OUT_SLAVE THEN
				fb_state_entry.i16_next_step := 50;
			ELSIF st_ecd_cmd.enu_cmd = CAM_SCALEING_SLAVE THEN
				fb_state_entry.i16_next_step := 60;
			ELSIF st_ecd_cmd.enu_cmd = READ_MOTION_POINT THEN
				fb_state_entry.i16_next_step := 70;
			ELSIF st_ecd_cmd.enu_cmd = WRITE_MOTION_POINT THEN
				fb_state_entry.i16_next_step := 80;
			ELSIF st_ecd_cmd.enu_cmd = READ_SLAVE_DYNAMICS THEN
				fb_state_entry.i16_next_step := 90;
			ELSIF st_ecd_cmd.enu_cmd = READ_CAMTABLE_CHAR THEN
				fb_state_entry.i16_next_step := 100;
			ELSIF st_ecd_cmd.enu_cmd = RESET THEN
				fb_state_entry.i16_next_step := 999;
			ELSE
				fb_state_entry.i16_next_step := 1000;
			END_IF
		END_IF

(*=======================================================*)
	20:	(* Gear in *)
		fb_ton_cmd_timeout.IN := TRUE;
		mc_gearindyn_axis.Enable := TRUE;
		IF mc_gearindyn_axis.Busy THEN
			fb_state_entry.i16_next_step := 22;
		END_IF

	22:
		IF mc_gearindyn_axis.InGear THEN
			mc_gearindyn_axis.Enable := FALSE;
			fb_state_entry.i16_next_step := 999;
		ELSIF mc_gearindyn_axis.Error THEN
			st_ecd_cmd.meldungen.sm_gear_in_slave := TRUE;
			err_id := mc_gearindyn_axis.ErrorID;
			fb_state_entry.i16_next_step := 1000;
		END_IF

		IF st_ecd_cmd.enu_cmd = GEAR_OUT_SLAVE THEN
			mc_gearindyn_axis.Enable := FALSE;
			fb_ton_cmd_timeout.IN := FALSE;
			fb_ton_vz.IN := FALSE;
			fb_state_entry.i16_next_step := 50;
		END_IF

(*=======================================================*)
	30:	(* Gear out *)
		fb_ton_cmd_timeout.IN := TRUE;
		mc_gearout_axis.Execute := TRUE;
		IF mc_gearout_axis.Busy THEN
			fb_state_entry.i16_next_step := 32;
		END_IF
	32:
		IF NOT mc_gearout_axis.Busy THEN
			mc_gearout_axis.Execute := FALSE;
			IF mc_gearout_axis.Done THEN
				fb_state_entry.i16_next_step := 999;
			ELSIF mc_gearout_axis.Error THEN
				st_ecd_cmd.meldungen.sm_gear_out_slave := TRUE;
				err_id := mc_gearout_axis.ErrorID;
				fb_state_entry.i16_next_step := 1000;
			END_IF
		END_IF

(*=======================================================*)
	40:	(* Cam in *)
		fb_ton_cmd_timeout.IN := NOT st_slaveachse.Status.CamTableQueued;
		mc_camin_axis.Execute := TRUE;
		IF mc_camin_axis.Busy THEN
			fb_state_entry.i16_next_step := 42;
		END_IF
		IF st_ecd_cmd.enu_cmd = CAM_OUT_SLAVE THEN
			mc_camin_axis.Execute := FALSE;
			fb_state_entry.i16_next_step := 50;
		END_IF
	42:
		fb_ton_cmd_timeout.IN := NOT st_slaveachse.Status.CamTableQueued;
		IF NOT mc_camin_axis.Busy THEN
			mc_camin_axis.Execute := FALSE;
			IF mc_camin_axis.InSync THEN
				fb_state_entry.i16_next_step := 999;
			ELSIF mc_camin_axis.Error THEN
				err_id := mc_camin_axis.ErrorID;
				mc_camin_axis.Execute := FALSE;
				st_ecd_cmd.meldungen.sm_cam_in_slave := TRUE;
				fb_state_entry.i16_next_step := 1000;
			END_IF
		END_IF

		IF st_ecd_cmd.enu_cmd = CAM_OUT_SLAVE THEN
			mc_camin_axis.Execute := FALSE;
			fb_ton_cmd_timeout.IN := FALSE;
			fb_ton_vz.IN := FALSE;
			fb_state_entry.i16_next_step := 50;
		END_IF

(*=======================================================*)
	50:	(* Cam out *)
		fb_ton_cmd_timeout.IN := TRUE;
		mc_camout_axis.Execute := TRUE;
		IF mc_camout_axis.Busy THEN
			fb_state_entry.i16_next_step := 52;
		END_IF
	52:
		IF NOT mc_camout_axis.Busy THEN
			mc_camout_axis.Execute := FALSE;
			IF mc_camout_axis.Done THEN
				fb_state_entry.i16_next_step := 999;
			ELSIF mc_camout_axis.Error THEN
				st_ecd_cmd.meldungen.sm_cam_out_slave := TRUE;
				err_id := mc_camout_axis.ErrorID;
				fb_state_entry.i16_next_step := 1000;
			END_IF
		END_IF

(*=======================================================*)
	60:	(* Cam scaleing *)
		fb_ton_cmd_timeout.IN := NOT st_slaveachse.Status.CamScalingPending;
		mc_cam_scaleing.Execute := TRUE;
		IF mc_cam_scaleing.Busy THEN
			fb_state_entry.i16_next_step := 62;
		END_IF
	62:
		fb_ton_cmd_timeout.IN := NOT st_slaveachse.Status.CamScalingPending;
		IF NOT mc_cam_scaleing.Busy THEN
			mc_cam_scaleing.Execute := FALSE;
			IF mc_cam_scaleing.Done THEN
				fb_state_entry.i16_next_step := 999;
			ELSIF mc_cam_scaleing.Error THEN
				st_ecd_cmd.meldungen.sm_cam_scaleing_slave := TRUE;
				err_id := mc_cam_scaleing.ErrorID;
				fb_state_entry.i16_next_step := 1000;
			END_IF
		END_IF

		IF st_ecd_cmd.enu_cmd = CAM_OUT_SLAVE THEN
			mc_cam_scaleing.Execute := FALSE;
			fb_ton_cmd_timeout.IN := FALSE;
			fb_ton_vz.IN := FALSE;
			fb_state_entry.i16_next_step := 50;
		END_IF

(*=======================================================*)
	70:	(* Lesen Motion Funktion Point *)
		fb_ton_cmd_timeout.IN := TRUE;
		mc_read_motion_function_point.Execute := TRUE;
		IF mc_read_motion_function_point.Busy THEN
			fb_state_entry.i16_next_step := 72;
		END_IF
	72:
		IF NOT mc_read_motion_function_point.Busy THEN
			mc_read_motion_function_point.Execute := FALSE;
			IF mc_read_motion_function_point.Done THEN
				fb_state_entry.i16_next_step := 999;
			ELSIF mc_read_motion_function_point.Error THEN
				st_ecd_cmd.meldungen.sm_read_motion_funktion_point := TRUE;
				err_id := mc_read_motion_function_point.ErrorID;
				fb_state_entry.i16_next_step := 1000;
			END_IF
		END_IF

(*=======================================================*)
	80:	(* Schreiben Motion Funktion Point *)
		fb_ton_cmd_timeout.IN := TRUE;
		mc_write_motion_function_point.Execute := TRUE;
		IF mc_write_motion_function_point.Busy THEN
			fb_state_entry.i16_next_step := 82;
		END_IF
	82:
		IF NOT mc_write_motion_function_point.Busy THEN
			mc_write_motion_function_point.Execute := FALSE;
			IF mc_write_motion_function_point.Done THEN
				fb_state_entry.i16_next_step := 999;
			ELSIF mc_write_motion_function_point.Error THEN
				st_ecd_cmd.meldungen.sm_write_motion_funktion_point := TRUE;
				err_id := mc_write_motion_function_point.ErrorID;
				fb_state_entry.i16_next_step := 1000;
			END_IF
		END_IF

(*=======================================================*)
	90:	(* Lesen der Slaveposition in einer Kurvenscheibe *)
		fb_ton_cmd_timeout.IN := TRUE;
		mc_read_camtable_slave_dynamics.Execute := TRUE;
		IF mc_read_camtable_slave_dynamics.Busy THEN
			fb_state_entry.i16_next_step := 92;
		END_IF
	92:
		IF NOT mc_read_camtable_slave_dynamics.Busy THEN
			mc_read_camtable_slave_dynamics.Execute := FALSE;
			IF mc_read_camtable_slave_dynamics.Done THEN
				fb_state_entry.i16_next_step := 999;
			ELSIF mc_read_camtable_slave_dynamics.Error THEN
				st_ecd_cmd.meldungen.sm_write_motion_funktion_point := TRUE;
				err_id := mc_read_camtable_slave_dynamics.ErrorID;
				fb_state_entry.i16_next_step := 1000;
			END_IF
		END_IF

(*=======================================================*)
	100:	(* Lesen der charakteristischen Werte einer Kurvenscheibe *)
		fb_ton_cmd_timeout.IN := TRUE;
		mc_read_camtable_characteristics.Execute := TRUE;
		IF mc_read_camtable_characteristics.Busy THEN
			fb_state_entry.i16_next_step := 102;
		END_IF
	102:
		IF NOT mc_read_camtable_characteristics.Busy THEN
			mc_read_camtable_characteristics.Execute := FALSE;
			IF mc_read_camtable_characteristics.Done THEN
				fb_state_entry.i16_next_step := 999;
			ELSIF mc_read_camtable_characteristics.Error THEN
				st_ecd_cmd.meldungen.sm_read_camtable_charakteristik := TRUE;
				err_id := mc_read_camtable_slave_dynamics.ErrorID;
				fb_state_entry.i16_next_step := 1000;
			END_IF
		END_IF

(*=======================================================*)
	999:	(* Ende - Befehl wurde korrekt abgearbeitet *)
		fb_ton_cmd_timeout.IN := FALSE;
		fb_ton_vz.IN := FALSE;

		mc_gearindyn_axis.Enable := FALSE;
		mc_gearout_axis.Execute := FALSE;
		mc_camin_axis.Execute := FALSE;
		mc_camout_axis.Execute := FALSE;
		mc_cam_scaleing.Execute := FALSE;
		mc_read_motion_function_point.Execute := FALSE;
		mc_write_motion_function_point.Execute := FALSE;
		mc_read_camtable_slave_dynamics.Execute := FALSE;
		mc_read_camtable_characteristics.Execute := FALSE;

		st_ecd_cmd.meldungen.sm_gear_in_slave := FALSE;
		st_ecd_cmd.meldungen.sm_gear_out_slave := FALSE;
		st_ecd_cmd.meldungen.sm_cam_in_slave := FALSE;
		st_ecd_cmd.meldungen.sm_cam_out_slave := FALSE;
		st_ecd_cmd.meldungen.sm_cam_scaleing_slave := FALSE;
		st_ecd_cmd.meldungen.sm_write_motion_funktion_point := FALSE;
		st_ecd_cmd.meldungen.sm_read_motion_funktion_point := FALSE;
		st_ecd_cmd.meldungen.sm_read_camtable_slave_dynamics := FALSE;
		st_ecd_cmd.meldungen.sm_read_camtable_charakteristik := FALSE;
		st_ecd_cmd.meldungen.sm_camgear_command_timeout := FALSE;

		fb_state_entry.i16_next_step := 10;

(*=======================================================*)
	1000: (* Fehler *)
		IF fb_state_entry.E THEN
			st_ecd_cmd.enu_cmd := NO_COMMAND;
			st_ecd_cmd.b_job_fehler := TRUE;
			fb_ton_cmd_timeout.IN := FALSE;
			fb_ton_vz.IN := FALSE;

			mc_gearindyn_axis.Enable := FALSE;
			mc_gearout_axis.Execute := FALSE;
			mc_camin_axis.Execute := FALSE;
			mc_camout_axis.Execute := FALSE;
			mc_cam_scaleing.Execute := FALSE;
			mc_read_motion_function_point.Execute := FALSE;
			mc_write_motion_function_point.Execute := FALSE;
			mc_read_camtable_slave_dynamics.Execute := FALSE;
			mc_read_camtable_characteristics.Execute := FALSE;
		END_IF

		(* Fehler reseten *)
		IF st_ecd_cmd.enu_cmd > ABORT THEN
			st_ecd_cmd.b_job_fehler := FALSE;

			st_ecd_cmd.meldungen.sm_gear_in_slave := FALSE;
			st_ecd_cmd.meldungen.sm_gear_out_slave := FALSE;
			st_ecd_cmd.meldungen.sm_cam_in_slave := FALSE;
			st_ecd_cmd.meldungen.sm_cam_out_slave := FALSE;
			st_ecd_cmd.meldungen.sm_cam_scaleing_slave := FALSE;
			st_ecd_cmd.meldungen.sm_write_motion_funktion_point := FALSE;
			st_ecd_cmd.meldungen.sm_read_motion_funktion_point := FALSE;
			st_ecd_cmd.meldungen.sm_read_camtable_slave_dynamics := FALSE;
			st_ecd_cmd.meldungen.sm_read_camtable_charakteristik := FALSE;
			st_ecd_cmd.meldungen.sm_camgear_command_timeout := FALSE;

			fb_state_entry.i16_next_step := 10;
			err_id :=0;
		END_IF
END_CASE

(* Timeout-Fehler aller Drivekommandos *)
IF fb_ton_cmd_timeout.Q THEN
	fb_ton_cmd_timeout.IN := FALSE;
	st_ecd_cmd.meldungen.sm_camgear_command_timeout := TRUE;
	fb_state_entry.i16_next_step := 1000;
END_IF

(* Statehistory *)
fb_state_entry(
	i16_next_step:= , 
	i16_pos:= 2,
	s_debugtext:= ,
	E=> ,
	X=> , 
	i16_step=> ,
	i16_last_step=> );

fb_cmd_history(i16_current_cmd:= st_ecd_cmd.enu_cmd, last_cmd=> );

(*=============================================================================================*)
(* Ab hier werden alle Cam und Gear Aufträge für eine Achse abgewickelt *)

(* Getriebegleichlauf an der Slaveachse einschalten *)
(* Alternativ kann der Getriebefaktor im Zähler als Fließkommawert angegeben werden, wenn der Nenner 1 ist. *)
mc_gearindyn_axis(
	Enable:= , 
	GearRatio:= r_getriebefaktor,
	Acceleration:= , 
	Deceleration:= , 
	Jerk:= , 
	BufferMode:= mc_buffermode_axis,
	Options:= , 
	Master:= st_masterachse,
	Slave:= st_slaveachse,
	InGear=> , 
	Busy=> , 
	Active=> , 
	CommandAborted=> , 
	Error=> , 
	ErrorID=> );

(*=============================================================================================*)
(* Getriebegleichlauf ausschalten *)
mc_gearout_axis(
	Execute:= ,
	Options:= ,
	Slave:= st_slaveachse,
	Done=> ,
	Busy=> ,
	Error=> ,
	ErrorID=> );

(*=============================================================================================*)
(* Kurvenscheibe am Slave aktivieren *)
mc_camin_axis(
	Execute:= , 
	ActivationMode:= mc_activation_mode_camin,
	ActivationPosition:= lr_activation_position_camin,
	CamTableID:= mc_cam_table_id,
	Scaling:= st_camscaling_data,
	Options:= st_camin_options,
	Master:= st_masterachse,
	Slave:= st_slaveachse,
	InSync=> , 
	Busy=> , 
	Active=> , 
	CommandAborted=> , 
	Error=> ,
	ErrorID=> );

(*=============================================================================================*)
(* Kurvenscheibe ausschalten *)
mc_camout_axis(
	Execute:= ,
	Slave:= st_slaveachse,
	Options:= ,
	Done=> ,
	Busy=> ,
	Error=> ,
	ErrorID=> );

(*=============================================================================================*)
(* Scalierung einer Kurvenscheibe *)
mc_cam_scaleing(
	Execute:= , 
	ActivationMode:= mc_activation_mode_scaleing,
	ActivationPosition:= lr_activation_position_scaleing,
	CamTableID:= mc_cam_table_id,
	Scaling:= st_camscaling_data,
	Options:= ,
	Slave:= st_slaveachse,
	Done=> , 
	Busy=> ,
	Active=> , 
	CommandAborted=> ,
	Error=> , 
	ErrorID=> );

(*=============================================================================================*)
(* Lesen eines Punktes in der Kurvenscheibe *)
mc_read_motion_function_point(
	Execute:= ,
	CamTableID:= mc_cam_table_id,
	PointID:= mc_cam_point_id,
	Point:= mc_motion_function_point,
	Done=> , 
	Busy=> , 
	Error=> , 
	ErrorID=> );

(*=============================================================================================*)
(* Verändern von einem Punkt in der Kurvenscheibe *)
mc_write_motion_function_point(
	Execute:= , 
	CamTableID:= mc_cam_table_id,
	PointID:= mc_cam_point_id,
	Point:= mc_motion_function_point,
	Done=> , 
	Busy=> , 
	Error=> ,
	ErrorID=> );

(*=============================================================================================*)
(* Lesen einer Slaveposition in der Kurvenscheibe *)
mc_read_camtable_slave_dynamics(
	Execute:= ,
	CamTableID:= mc_cam_table_id,
	MasterPosition:= r_master_position,
	Done=> , 
	Busy=> ,
	Error=> , 
	ErrorID=> ,
	SlavePosition=> , 
	SlaveVelocity=> , 
	SlaveAcceleration=> );

(*=============================================================================================*)
(* Lesen der charakteristischen Werte einer Kurvenscheibe *)
mc_read_camtable_characteristics(
	Execute:= , 
	CamTableID:= mc_cam_table_id,
	CamTableCharac:= st_cam_table_characteristics,
	Done=> , 
	Busy=> , 
	Error=> , 
	ErrorID=> );
END_FUNCTION_BLOCK

(* POU EPT Lib/Funktionsbausteine/ST_Taktzeit, ST *)
FUNCTION_BLOCK ST_Taktzeit
VAR_INPUT
	b_start			: BOOL;
END_VAR
VAR_OUTPUT
	t_zeit			: TIME;
END_VAR
VAR
	fb_f_trig_stop		: F_TRIG;
	fb_ton			: TON;
END_VAR
fb_f_trig_stop(CLK:= b_start, Q=> );

IF fb_f_trig_stop.Q THEN
	t_zeit := fb_ton.ET;
END_IF

fb_ton(IN:= b_start, PT:= t#20h, Q=> );
END_FUNCTION_BLOCK

(* POU Gemeinsamkeiten17xx/Visu/ST_Message_Produktion, ST *)
PROGRAM ST_Message_Produktion
VAR_INPUT
	b_PM_Quitt		:BOOL:=FALSE;
END_VAR
VAR
	LockFlag				: BOOL := FALSE;	(* Ganz wichtig, wenn diese Variable TRUE ist, dann kann die Struktur "Visu.MeldungProduktion" nicht verändert werden *)
	b_init					: BOOL:=FALSE;

	fb_r_trig_LockFree		: R_TRIG;
	fb_f_trig_Button1		: F_TRIG;
	fb_f_trig_Button2		: F_TRIG;
	fb_ton_quitt			: TON;
	fb_ton_autoquitt		: TON;

	i						: INT;
END_VAR
IF NOT b_init THEN
	b_init:=TRUE;
END_IF


(*Zeiten*)
fb_ton_quitt(IN:= b_PM_Quitt, PT:= T#100ms, Q=> , ET=> );
fb_ton_autoquitt(IN:= Visu.MeldungProduktion.Name='' AND LockFlag , PT:= T#5000ms, Q=> , ET=> );

(*Flanken*)
fb_f_trig_Button1(CLK:= Visu.MeldungProduktion.Button1.tasten, Q=> );	(* OK *)
fb_f_trig_Button2(CLK:= Visu.MeldungProduktion.Button2.tasten, Q=> );	(* Cancel *)

fb_r_trig_LockFree(CLK:= fb_f_trig_Button1.Q OR	(* OK *)
						fb_f_trig_Button2.Q OR	(* Cancel *)
						fb_ton_quitt.Q, Q=> );

IF fb_r_trig_LockFree.Q OR
	fb_ton_autoquitt.Q THEN
	Visu.MeldungProduktion.Color_R:=0;
	Visu.MeldungProduktion.Color_G:=0;
	Visu.MeldungProduktion.Color_B:=0;
	Visu.MeldungProduktion.Name:='';
	Visu.MeldungProduktion.Button1.sichtbar:=FALSE;
	Visu.MeldungProduktion.Button1.Text:='';
	Visu.MeldungProduktion.Button2.sichtbar:=FALSE;
	Visu.MeldungProduktion.Button2.Text:='';
	ClearMessageLines();
	visu.MeldungProduktion.ShowMessage:=FALSE;
	b_PM_Quitt:=FALSE;
	LockFree();
END_IF


(* wenn etwas in Name drin steht, dann soll Meldung angezeigt werden *)
IF	Visu.MeldungProduktion.Name <> '' THEN
	visu.MeldungProduktion.ShowMessage:=TRUE;
END_IF

(*
Beispiel Aufruf

(*=======================================================*)
	900:	(*Warten bis keine andere Produktions Meldung ansteht *)
	
		(*-----------------------Weiterschaltbedingungen----------------------------*)
		IF TestAndSet(ST_Message_Produktion.LockFlag) THEN
			ST_Message_Produktion.ClearMessageLines();
			fb_state_entry.i16_next_step := 910;
		END_IF
		
(*=======================================================*)
	910:  (*Produktions Meldung *)
		IF fb_state_entry.E THEN
			Visu.MeldungProduktion.Color:=Color.yellow;
			Visu.MeldungProduktion.Name:='';
			Visu.MeldungProduktion.Text:='PM100';
	
			Visu.MeldungProduktion.Button1.unsichtbar:=FALSE;	(*OK*)
			Visu.MeldungProduktion.Button2.unsichtbar:=FALSE;	(*Cancel*)
		END_IF

		(*-----------------------Weiterschaltbedingungen----------------------------*)
		IF ST_Message_Produktion.fb_f_trig_Button1.Q THEN
			fb_state_entry.i16_next_step:=920;
		ELSIF ST_Message_Produktion.fb_f_trig_Button2.Q THEN
			fb_state_entry.i16_next_step:=FEHLER;
		ELSIF b_Help THEN
			ST_Message_Produktion.b_PM_Quitt := TRUE;
			fb_state_entry_2.i16_next_step:=BEREIT;
		END_IF

		---WICHTIG---
		Die Variable "ST_Message_Produktion.b_PM_Quitt" darf nicht auf FALSE gesetzt werden.
		Das wird im Baustein ST_Message_Produktion gemacht.

*)
END_PROGRAM
ACTION ClearMessageLines:
FOR i:=0 TO 9 DO
	Visu.MeldungProduktion.Text[i]:='';
END_FOR;
END_ACTION
ACTION LockFree:
LockFlag := FALSE;	(* wieder freigeben *)
END_ACTION

(* POU Gemeinsamkeiten17xx/Achsen/ST_Y_Achse, ST *)
PROGRAM ST_Y_Achse
VAR_INPUT
	st_config_achse						: struct_ecd_config;
	st_ctrl_in								: struct_ctrl_in;
	e_steuerung_ein						: BOOL;
	e_ba_mit_bedingungen				: BOOL;
	e_tuere_vorne_offen					: BOOL;
	e_tuere_hinten_offen					: BOOL;
	e_not_steu_tuer_schutz_ok				: BOOL;
	lr_tmp_Achspos						: LREAL;

	b_start_in							: BOOL;
	lr_Achspos_in						: LREAL;
	lr_Velo_in							: LREAL;
	enu_cmd_in							: enum_ecd_cmd;
END_VAR
VAR_IN_OUT
	st_visu								: struct_ecd_visu;
END_VAR
VAR_OUTPUT
	st_ctrl_out							: struct_ctrl_out;
	lr_RecPos							: LREAL;
END_VAR
VAR
	st_sm						 		: struct_ecd_meldungen;
	st_drive_cmd							: struct_ecd_cmd;
	fb_ton_wz							: TON;
	fb_ton_quitt							: TON;
	fb_ton_wz_disable						: TON;
	fb_r_trig_start							: R_TRIG;
	fb_r_trig_start_in						: R_TRIG;
	fb_r_trig_taste_plus					: R_TRIG;
	fb_r_trig_taste_minus					: R_TRIG;
	fb_r_trig_hand_dialog					: R_TRIG;
	fb_axis								: ST_AxisJobCtrl_Motion;
	fb_state_entry							: ST_StateEntry;
	fb_ton_uez							: TON;
	fb_ton_regelfreigabe_y_achse			: TON;
	i									: UINT := 0;
	lr_pos_ohneverschiebung			: LREAL;
	fb_r_trig_limit_sensor_positiv			: R_TRIG;
	fb_r_trig_limit_sensor_negativ			: R_TRIG;
	fb_r_trig_skalierungsnocken				: R_TRIG;
	fb_r_trig_nullpunkt_setzen				: R_TRIG;

	b_hand_dialog_aktiv					: BOOL := FALSE;
	sm_kein_nocken_definiert				: BOOL := FALSE;

	st_geschwindigkeiten					: struct_ecd_geschwindigkeiten;
	e_referenz_sensor						AT %I* : BOOL;
	i16_torque							AT %I* : INT;
	i16_DigitalInput						AT %I* : INT;

	lr_decceleration_nothalt				: LREAL;
	lr_decceleration_normal				: LREAL;

	i16_state_msg						: INT;
	lr_MaxSoftPosLimit					:LREAL;
	lr_MinSoftPosLimit						:LREAL;
	b_EndlageErreicht						:BOOL;
	fb_r_trig_Endlage						: R_TRIG;
END_VAR
(* Zeiten *)
fb_ton_wz(IN:= , PT:= , Q=>  , ET=> );
fb_ton_uez(IN:= , PT:= , Q=>  , ET=> );
fb_ton_quitt(IN:= , PT:= t#100ms, Q=> , ET=> );
fb_ton_wz_disable(IN:= , PT:= t#500ms, Q=> , ET=> );

(* Flanken *)
fb_r_trig_limit_sensor_positiv(CLK:= st_config_achse.b_limitsensor_positiv_vorhanden AND NOT fb_axis.e_limit_sensor_positive, Q=> );
fb_r_trig_limit_sensor_negativ(CLK:= st_config_achse.b_limitsensor_negativ_vorhanden AND NOT fb_axis.e_limit_sensor_negative, Q=> );
fb_r_trig_taste_plus(CLK:= ST_Euchner_Handbedienpult.b_Taste_Plus, Q=> );
fb_r_trig_taste_minus(CLK:= ST_Euchner_Handbedienpult.b_Taste_Minus, Q=> );
fb_r_trig_start(CLK:= st_ctrl_in.b_start, Q=> );
fb_r_trig_start_in(CLK:= b_start_in, Q=> );
fb_r_trig_skalierungsnocken(CLK:= nockenschaltwerk_bestueckachse.fb.arr_spur[SP_START_SKALIERUNG], Q=> );
fb_r_trig_hand_dialog(CLK:= b_hand_dialog_aktiv, Q=> );
fb_r_trig_nullpunkt_setzen(CLK:=axis_y_achse.st_visu.b_nullpunkt_setzen);

(* Achse steuern *)
fb_axis(
	e_referenznocken:= ,
	b_refsensor_vorhanden:= st_config_achse.b_refsensor_vorhanden,
	b_limitsensor_positiv_vorhanden:= st_config_achse.b_limitsensor_positiv_vorhanden,
	b_limitsensor_negativ_vorhanden:= st_config_achse.b_limitsensor_negativ_vorhanden,
	i16_achstyp := st_config_achse.i16_achstyp,
	lr_override_vorgabe:= ST_TippTasten.lr_override,
	st_position:= ,
	mc_richtung_modulo:= ,
	mc_richtung_velocity:= ,
	mc_referenzmodus:= ,
	mc_buffermode_axis:= ,
	ui16_soeparam_write_value:= ,
	w_idn:= ,
	i16_nc_parameter_nummer:= ,
	r_wert_nc_write_parameter:= ,
	st_vorgabe_geschwindigkeiten:= st_geschwindigkeiten,
	lr_soll_geschwindigkeit:= ,
	b_bedingung_sls:= NOT e_tuere_vorne_offen OR NOT e_tuere_hinten_offen,
	st_ads_info := ,
	st_eccoe_sdo := ,
	st_masterachse:= y_achse,
	st_visu_axis:= st_visu,
	st_ecd_cmd:= st_drive_cmd,
	ui16_soeparam_read_value=> ,
	r_wert_nc_read_parameter=>  ,
	lr_RecPos=> lr_RecPos,
	b_TriggerInput:=i16_DigitalInput.2,
	b_FallingEdge:=TRUE);

(* Achse mit dem Euchner Handbediengerät vorwärts und rückwärts Bewegen*)
IF gi16_betriebsart = HAND AND fb_r_trig_hand_dialog.Q THEN
	fb_state_entry.i16_next_step := HANDRAD;
END_IF

IF gi16_betriebsart = HAND THEN
	(* Button in der Oberfläche zum setzen des Nullpunktes *)
	IF fb_r_trig_nullpunkt_setzen.Q THEN
		fb_state_entry.i16_next_step :=	NULLPUNKT_SETZEN;
	END_IF
END_IF


(*Meldung Achse hat Endlage überfahren*)
IF lr_MinSoftPosLimit<>0 AND
 lr_MinSoftPosLimit > gst_datensatz.st_md.st_md_y_achse.lr_wt_uebergabepos THEN
	b_EndlageErreicht:=TRUE;
ELSE
	b_EndlageErreicht:=FALSE;
END_IF

fb_r_trig_Endlage(CLK:= b_EndlageErreicht , Q=> );

IF fb_r_trig_Endlage.Q THEN
	i16_state_msg := 1;
END_IF

(*Produktionsmeldung für Endlage überfahren*)
CASE i16_state_msg OF
	1: (*Warten bis keine ander Produktions Meldung ansteht *)
		IF	TestAndSet(ST_Message_Produktion.LockFlag) THEN
			ST_Message_Produktion.ClearMessageLines();
			i16_state_msg := 2;
		END_IF

